(* IEC 61131-3 sources: std_i2980_v2.06_cp053/Source/IMM/ieccontrol/MoldHeightAdjust1 (part 3) *)

(* ---- ABAdjustPositionChange.pu ---- *)
(*
@h    ! WARNING !
@h    The Kemro K2 system (including software) only meets category B according to EN 954-1,
@h    thus it is not intended for usage in safety-relevant control applications in the field
@h    of personal safety (e.g. emergency stop).
@h    To implement potentially necessary safety-relevant control tasks, always use additional
@h    external safety devices that are intended for the particular purpose, and meet the necessary
@h    functional safety.
@h    For further information see EN 954-1 (EN ISO 13849-1) and/or the K2-x00 user manual, chapter
@h    "CE conformity, directives and standards".

This algo sends the mold height to a specified position by controlling the
Mold Height Movements.
*)

IMPORT_OVER_LISTFILE
 SET_ALARM
, cMoveFwd
, cMoveMoldHeight
, cMoveBwd
, tsMoldHeightPositions
, tsEndpointMonitor
, tevStartRequest
, tsDeviceId
, tevStartRequestData
, FBStop
, FBCheckReady
, tnMovementDirection

END_IMPORT

ALGORITHM_BLOCK ABAdjustPositionChange #DUMMY_EDIT_BLOCK

SYSTEM_VAR
 sv_MoldHeightPositions : tsMoldHeightPositions;
 sv_MoldHeightEndpoints : tsEndpointMonitor;
 sv_rActMoldHeightPosition : REAL;
 sv_iThisStepsSetImpulses : UDINT;
 sv_rDistancePerImpulse : REAL;
END_VAR

SYSTEM_OBJECT
 evStartRequest : tevStartRequest;
 erMoldHeightAdjustAborted : ALARM;
 erMoldHeightAdjustFinished : ALARM;
END_OBJECT

(*
This algo controls the mold height automatic position change:
- A desired position is set on the hmi. By starting the automatic mold height adjustment this algo is called.
- The desired position is translated into a number of increments and direction to move to.
- The movement is started until the position reached flags are set by the movements of MoldHeight1.
- The ready flag is set and the algo won't be called any more.
*)

ALGORITHM aRun

VAR_INPUT
 bStop : BOOL;
END_VAR

VAR_OUTPUT
 bReady : BOOL;
END_VAR

VAR_INPUT
 DeviceIdMoldHeight : tsDeviceId;
END_VAR

VAR
 iTempImpulses : INT;
 evStartRequestData : tevStartRequestData;
 fbStop : FBStop;
 fbCheckReady : FBCheckReady;
 MovementDirection : tnMovementDirection;
END_VAR

(* IecGraph-Code *)

(* init step *)
INITIAL_STEP START:
END_STEP

(* steps *)
STEP PREPARE_MOVEMENT:
aPrepareMovement (P);
END_STEP

STEP MOVE:
AReset (P);
END_STEP

ACTION AReset: #BEGIN_EDIT_BLOCK
sv_MoldHeightEndpoints.bPositionForStepReached := FALSE;

;#END_EDIT_BLOCK END_ACTION (*AReset*)
STEP MOVE_FWD_TO_POS:
aMoveFwdToPos (P);
aCheckFwdReady (N);
END_STEP

STEP MOVE_BWD_TO_POS:
aMoveBwdToPos (P);
aCheckBwdReady (N);
END_STEP

STEP READY:
ResetMovementFlags (P);
END_STEP

ACTION ResetMovementFlags: #BEGIN_EDIT_BLOCK
IF bStop THEN
    //stop active device
    fbStop(DeviceId := DeviceIdMoldHeight);
END_IF;

IF sv_MoldHeightEndpoints.bPositionForStepReached THEN
    SET_ALARM(erMoldHeightAdjustFinished);
ELSE
    SET_ALARM(erMoldHeightAdjustAborted);
END_IF;

bReady := TRUE;

;#END_EDIT_BLOCK END_ACTION (*ResetMovementFlags*)

(* transitions *)
GO_ON_TRANSITION StartTrans FROM START TO PREPARE_MOVEMENT :=  #BEGIN_EDIT_BLOCK
TRUE
;#END_EDIT_BLOCK
END_TRANSITION

GO_ON_TRANSITION TAdjust FROM PREPARE_MOVEMENT TO MOVE :=  #BEGIN_EDIT_BLOCK
iTempImpulses <> 0
;#END_EDIT_BLOCK
END_TRANSITION

GO_ON_TRANSITION TNoAdjustNeeded FROM PREPARE_MOVEMENT TO READY :=  #BEGIN_EDIT_BLOCK
iTempImpulses = 0
;#END_EDIT_BLOCK
END_TRANSITION

GO_ON_TRANSITION CheckMovementDirection1 FROM MOVE TO MOVE_FWD_TO_POS :=  #BEGIN_EDIT_BLOCK
MovementDirection = nForward
;#END_EDIT_BLOCK
END_TRANSITION

TRANSITION CheckMovementFinished1 FROM MOVE_FWD_TO_POS TO READY :=  #BEGIN_EDIT_BLOCK
fbCheckReady.bReady OR bStop
;#END_EDIT_BLOCK
END_TRANSITION

GO_ON_TRANSITION CheckMovementDirection2 FROM MOVE TO MOVE_BWD_TO_POS :=  #BEGIN_EDIT_BLOCK
MovementDirection = nBackward
;#END_EDIT_BLOCK
END_TRANSITION

TRANSITION CheckMovementFinished2 FROM MOVE_BWD_TO_POS TO READY :=  #BEGIN_EDIT_BLOCK
fbCheckReady.bReady OR bStop
;#END_EDIT_BLOCK
END_TRANSITION

TRANSITION TLoopBack FROM READY TO START :=  #BEGIN_EDIT_BLOCK
TRUE
;#END_EDIT_BLOCK
END_TRANSITION

(* end IecGraph-Code *)
(* sfc-code *)

(* stand alone actions *)
ACTION aMoveFwdToPos: #BEGIN_EDIT_BLOCK
(*@ MoldHeightAdjustN.ABAdjustPositionChange.aMoveFwdToPos.Start the mold height forward movement.*)
evStartRequestData.DeviceId := DeviceIdMoldHeight;
evStartRequestData.MoveDir := cMoveFwd;
evStartRequestData.MoveId := cMoveFwd;
SET_EVENT(evStartRequest, evStartRequestData);

;#END_EDIT_BLOCK END_ACTION (*aMoveFwdToPos*)
ACTION aMoveBwdToPos: #BEGIN_EDIT_BLOCK
(*@ MoldHeightAdjustN.ABAdjustPositionChange.aMoveBwdToPos.Start the mold height backwar movement.*)
evStartRequestData.DeviceId := DeviceIdMoldHeight;
evStartRequestData.MoveDir := cMoveBwd;
evStartRequestData.MoveId := cMoveBwd;
SET_EVENT(evStartRequest, evStartRequestData);

;#END_EDIT_BLOCK END_ACTION (*aMoveBwdToPos*)
ACTION aPrepareMovement: #BEGIN_EDIT_BLOCK

(*@ MoldHeightAdjustN.ABAdjustPositionChange.aPrepareMovement.Reset the CalcFinished and AutoAdjustFinished flag
                                                for normal operation.*)
bReady := FALSE;

(*@ MoldHeightAdjustN.ABAdjustPositionChange.aPrepareMovement.Calculate the number of Impulses the mold height
                                                should move like this:
                                                Distance = Actual Position - MoveTo Position;
                                                Impulses To Move = Distance / Distance per Impulse*)
IF sv_rDistancePerImpulse > 0.0 THEN
   //avoid division by zero
   iTempImpulses := REAL_TO_INT((sv_rActMoldHeightPosition - sv_MoldHeightPositions.rMoveToMoldHeightPosition)/sv_rDistancePerImpulse);
ELSE
   iTempImpulses := 0;
END_IF;

(*@ MoldHeightAdjustN.ABAdjustPositionChange.aPrepareMovement.Check if the position as the same as the actual
                                                position and stop the movement if it so.
                                                Else check/set the direction. Negative number of Impulses to Move
                                                means Move Backward (If so, remove the negative sign of Impulses
                                                to Move.*)
IF iTempImpulses = 0 THEN
    bReady := TRUE;
ELSIF iTempImpulses < 0 THEN
    MovementDirection := nBackward;
    iTempImpulses := ABS(iTempImpulses);
ELSIF iTempImpulses > 0 THEN
    MovementDirection := nForward;
END_IF;

(*@ MoldHeightAdjustN.ABAdjustPositionChange.aPrepareMovement.Set the system variable for impulses to move*)
sv_iThisStepsSetImpulses := INT_TO_UDINT(iTempImpulses);

;#END_EDIT_BLOCK END_ACTION (*aPrepareMovement*)
ACTION aCheckFwdReady: #BEGIN_EDIT_BLOCK
(**************************************** WARNING ********************************************
 *** The KEBA Kemro K2 System including software is not intended for safety control tasks! ***
 ***                       For further information see Comment tab!                        ***
 *********************************************************************************************)

fbCheckReady(DeviceId := DeviceIdMoldHeight);

;#END_EDIT_BLOCK END_ACTION (*aCheckFwdReady*)
ACTION aCheckBwdReady: #BEGIN_EDIT_BLOCK
(**************************************** WARNING ********************************************
 *** The KEBA Kemro K2 System including software is not intended for safety control tasks! ***
 ***                       For further information see Comment tab!                        ***
 *********************************************************************************************)

fbCheckReady(DeviceId := DeviceIdMoldHeight);

;#END_EDIT_BLOCK END_ACTION (*aCheckBwdReady*)
(* end sfc-code *)

END_ALGORITHM

END_ALGORITHM_BLOCK

#END_OF_IEC_PART

@Puma @IecEditor 6 68 @Pou 25
@@@BEG_Comment@@@
@h    ! WARNING !
@h    The Kemro K2 system (including software) only meets category B according to EN 954-1,
@h    thus it is not intended for usage in safety-relevant control applications in the field
@h    of personal safety (e.g. emergency stop).
@h    To implement potentially necessary safety-relevant control tasks, always use additional
@h    external safety devices that are intended for the particular purpose, and meet the necessary
@h    functional safety.
@h    For further information see EN 954-1 (EN ISO 13849-1) and/or the K2-x00 user manual, chapter
@h    "CE conformity, directives and standards".

This algo sends the mold height to a specified position by controlling the
Mold Height Movements.
@@@END_Comment@@@

@BEG_Contents

@BEG_Func
@RT(17)FuncTreeContainer
1
@Var @RT(9)SET_ALARM @RT(0) @T @T @DERIVED 0 @F @RT(23)KEBA_STANDARD_PROCEDURE @F
@T
@BEG_Attrib
0 @RT(0) @RT(0)
@END_Attrib
1 1 @F @F @F @F

@END_Func

@BEG_Const
@RT(18)ConstTreeContainer
3
@Var @RT(8)cMoveFwd @RT(0) @T @F @DT @RT(4)DINT @RT(0) @T @T @BASIC 0 @F
@F @F
@T
@BEG_Attrib
0 @RT(2)12 @RT(16)movement forward
@END_Attrib
1 1 @F @F @F @F

@Var @RT(15)cMoveMoldHeight @RT(0) @T @F @DT @RT(4)DINT @RT(0) @T @T @BASIC 0 @F
@F @F
@T
@BEG_Attrib
0 @RT(2)29 @RT(23)movement of mold height
@END_Attrib
1 1 @F @F @F @F

@Var @RT(8)cMoveBwd @RT(0) @T @F @DT @RT(4)DINT @RT(0) @T @T @BASIC 0 @F
@F @F
@T
@BEG_Attrib
0 @RT(2)11 @RT(17)movement backward
@END_Attrib
1 1 @F @F @F @F

@END_Const

@BEG_Export

@BEG_Kind
@ALGORITHM_BLOCK @RT(22)ABAdjustPositionChange @STRUCTURED_TEXT
@RT(0) @RT(0) @RT(0)
@END_Kind

@BEG_Dcl
@RT(16)DclTreeContainer
8
@Var @RT(22)sv_MoldHeightPositions @RT(0) @T @T @DERIVED 0 @T @T @DT @RT(21)tsMoldHeightPositions @RT(0) @T @T @UNKNOWN 0 @F
@F @F
@T
@BEG_Attrib
3 @RT(0) @RT(0) @RT(0)
@END_Attrib
1 8 @F @F @F @F

@Var @RT(22)sv_MoldHeightEndpoints @RT(0) @T @T @DERIVED 0 @T @T @DT @RT(17)tsEndpointMonitor @RT(0) @T @T @UNKNOWN 0 @F
@F @F
@T
@BEG_Attrib
3 @RT(0) @RT(0) @RT(0)
@END_Attrib
1 8 @F @F @F @F

@Var @RT(25)sv_rActMoldHeightPosition @RT(0) @T @F @DT @RT(4)REAL @RT(0) @T @T @BASIC 0 @F
@F @F
@T
@BEG_Attrib
3 @RT(0) @RT(0) @RT(0)
@END_Attrib
1 8 @F @F @F @F

@Var @RT(24)sv_iThisStepsSetImpulses @RT(0) @T @F @DT @RT(5)UDINT @RT(0) @T @T @BASIC 0 @F
@F @F
@T
@BEG_Attrib
3 @RT(0) @RT(0) @RT(0)
@END_Attrib
1 8 @F @F @F @F

@Var @RT(22)sv_rDistancePerImpulse @RT(0) @T @F @DT @RT(4)REAL @RT(0) @T @T @BASIC 0 @F
@F @F
@T
@BEG_Attrib
3 @RT(0) @RT(0) @RT(0)
@END_Attrib
1 8 @F @F @F @F

@Var @RT(14)evStartRequest @RT(0) @T @T @DERIVED 0 @T @T @DT @RT(15)tevStartRequest @RT(0) @T @T @UNKNOWN 0 @F
@F @F
@T
@BEG_Attrib
3 @RT(0) @RT(0) @RT(0)
@END_Attrib
1 7 @F @F @F @F

@Var @RT(25)erMoldHeightAdjustAborted @RT(0) @T @F @DT @RT(5)ALARM @RT(0) @T @T @BASIC 0 @F
@F @F
@T
@BEG_Attrib
3 @RT(0) @RT(0) @RT(0)
@END_Attrib
1 7 @F @F @F @F

@Var @RT(26)erMoldHeightAdjustFinished @RT(0) @T @F @DT @RT(5)ALARM @RT(0) @T @T @BASIC 0 @F
@F @F
@T
@BEG_Attrib
3 @RT(0) @RT(0) @RT(0)
@END_Attrib
1 7 @F @F @F @F

@END_Dcl

@END_Export

@BEG_Body

1

@BEG_Export

@BEG_Algo
@ALGORITHM @RT(4)aRun @SEQUENTIAL_FLOW_CHART
@RT(0) @RT(0) @RT(0) @F @F
@END_Algo

@BEG_Dcl
@RT(16)DclTreeContainer
8
@Var @RT(5)bStop @RT(0) @T @F @DT @RT(4)BOOL @RT(0) @T @T @BASIC 0 @F
@F @F
@T
@BEG_Attrib
3 @RT(0) @RT(0) @RT(0)
@END_Attrib
1 1 @F @F @F @F

@Var @RT(6)bReady @RT(0) @T @F @DT @RT(4)BOOL @RT(0) @T @T @BASIC 0 @F
@F @F
@T
@BEG_Attrib
3 @RT(0) @RT(0) @RT(0)
@END_Attrib
1 3 @F @F @F @F

@Var @RT(18)DeviceIdMoldHeight @RT(0) @T @T @DERIVED 0 @T @T @DT @RT(10)tsDeviceId @RT(0) @T @T @UNKNOWN 0 @F
@F @F
@T
@BEG_Attrib
3 @RT(0) @RT(0) @RT(0)
@END_Attrib
1 1 @F @F @F @F

@Var @RT(13)iTempImpulses @RT(0) @T @F @DT @RT(3)INT @RT(0) @T @T @BASIC 0 @F
@F @F
@T
@BEG_Attrib
3 @RT(0) @RT(0) @RT(0)
@END_Attrib
1 0 @F @F @F @F

@Var @RT(18)evStartRequestData @RT(0) @T @T @DERIVED 0 @T @T @DT @RT(19)tevStartRequestData @RT(0) @T @T @UNKNOWN 0 @F
@F @F
@T
@BEG_Attrib
3 @RT(0) @RT(0) @RT(0)
@END_Attrib
1 0 @F @F @F @F

@Var @RT(6)fbStop @RT(0) @T @T @DERIVED 0 @T @T @DT @RT(6)FBStop @RT(0) @T @T @UNKNOWN 0 @F
@F @F
@T
@BEG_Attrib
3 @RT(0) @RT(0) @RT(0)
@END_Attrib
1 0 @F @F @F @F

@Var @RT(12)fbCheckReady @RT(0) @T @T @DERIVED 0 @T @T @DT @RT(12)FBCheckReady @RT(0) @T @T @UNKNOWN 0 @F
@F @F
@T
@BEG_Attrib
3 @RT(0) @RT(0) @RT(0)
@END_Attrib
1 0 @F @F @F @F

@Var @RT(17)MovementDirection @RT(0) @T @T @DERIVED 0 @T @T @DT @RT(19)tnMovementDirection @RT(0) @T @T @UNKNOWN 0 @F
@F @F
@T
@BEG_Attrib
3 @RT(0) @RT(0) @RT(0)
@END_Attrib
1 0 @F @F @F @F

@END_Dcl

@END_Export

@BEG_SfcBody
17 12 14

@BEG_SfcData 2
@StepSeq @RT(4)sseq @F 1
@Loop @RT(4)loop @F 2
@StepSeq @RT(3)seq @F 7
@Step @RT(5)START @F @T @F @F @RT(0) @F
@AcbCont @RT(7)unnamed @F 0

@Trans @RT(10)StartTrans @F @T @F @F @T @F @TL(2)
TRUE

@RT(6)Trans1 @F
@Step @RT(16)PREPARE_MOVEMENT @F @F @F @F @RT(0) @F
@AcbCont @RT(7)unnamed @F 1
@Acb @RT(16)aPrepareMovement @F @F @RT(1)P @RT(0) @F @F @T @F

@AltBranch @RT(3)alt @F 2
@TransSeq @RT(4)tseq @F 1
@Trans @RT(7)TAdjust @F @T @F @F @T @F @TL(2)
iTempImpulses <> 0

@RT(6)Trans2 @F

@TransSeq @RT(4)tseq @F 2
@Trans @RT(15)TNoAdjustNeeded @F @T @F @F @T @F @TL(2)
iTempImpulses = 0

@RT(7)Trans13 @F
@Goto @RT(5)READY @F @F

@Step @RT(4)MOVE @F @F @F @F @RT(0) @F
@AcbCont @RT(7)unnamed @F 1
@Acb @RT(6)AReset @F @T @RT(1)P @RT(0) @F @F @T @TL(2)
sv_MoldHeightEndpoints.bPositionForStepReached := FALSE;

@F

@AltBranch @RT(3)alt @F 2
@TransSeq @RT(4)tseq @F 3
@Trans @RT(23)CheckMovementDirection1 @F @T @F @F @T @F @TL(2)
MovementDirection = nForward

@RT(6)Trans3 @F
@Step @RT(15)MOVE_FWD_TO_POS @F @F @F @F @RT(0) @F
@AcbCont @RT(7)unnamed @F 2
@Acb @RT(13)aMoveFwdToPos @F @F @RT(1)P @RT(0) @F @F @T @F
@Acb @RT(14)aCheckFwdReady @F @F @RT(1)N @RT(0) @F @F @F @F

@Trans @RT(22)CheckMovementFinished1 @F @T @F @F @T @T @TL(2)
fbCheckReady.bReady OR bStop

@RT(6)Trans5 @F

@TransSeq @RT(4)tseq @F 3
@Trans @RT(23)CheckMovementDirection2 @F @T @F @F @T @F @TL(2)
MovementDirection = nBackward

@RT(6)Trans4 @F
@Step @RT(15)MOVE_BWD_TO_POS @F @F @F @F @RT(0) @F
@AcbCont @RT(7)unnamed @F 2
@Acb @RT(13)aMoveBwdToPos @F @F @RT(1)P @RT(0) @F @F @F @F
@Acb @RT(14)aCheckBwdReady @F @F @RT(1)N @RT(0) @F @F @F @F

@Trans @RT(22)CheckMovementFinished2 @F @T @F @F @T @T @TL(2)
fbCheckReady.bReady OR bStop

@RT(6)Trans5 @F

@Step @RT(5)READY @F @F @T @F @RT(0) @F
@AcbCont @RT(7)unnamed @F 1
@Acb @RT(18)ResetMovementFlags @F @T @RT(1)P @RT(0) @F @F @T @TL(13)
IF bStop THEN
    //stop active device
    fbStop(DeviceId := DeviceIdMoldHeight);
END_IF;

IF sv_MoldHeightEndpoints.bPositionForStepReached THEN
    SET_ALARM(erMoldHeightAdjustFinished);
ELSE
    SET_ALARM(erMoldHeightAdjustAborted);
END_IF;

bReady := TRUE;

@F

@Trans @RT(9)TLoopBack @F @T @T @T @T @T @TL(2)
TRUE

@RT(6)Trans7 @F

@END_SfcData
@SaActions 5
@SaText @RT(13)aMoveFwdToPos 1 @TL(6)
(*@ MoldHeightAdjustN.ABAdjustPositionChange.aMoveFwdToPos.Start the mold height forward movement.*)
evStartRequestData.DeviceId := DeviceIdMoldHeight;
evStartRequestData.MoveDir := cMoveFwd;
evStartRequestData.MoveId := cMoveFwd;
SET_EVENT(evStartRequest, evStartRequestData);

@SaText @RT(13)aMoveBwdToPos 1 @TL(6)
(*@ MoldHeightAdjustN.ABAdjustPositionChange.aMoveBwdToPos.Start the mold height backwar movement.*)
evStartRequestData.DeviceId := DeviceIdMoldHeight;
evStartRequestData.MoveDir := cMoveBwd;
evStartRequestData.MoveId := cMoveBwd;
SET_EVENT(evStartRequest, evStartRequestData);

@SaText @RT(16)aPrepareMovement 1 @TL(33)

(*@ MoldHeightAdjustN.ABAdjustPositionChange.aPrepareMovement.Reset the CalcFinished and AutoAdjustFinished flag
                                                for normal operation.*)
bReady := FALSE;

(*@ MoldHeightAdjustN.ABAdjustPositionChange.aPrepareMovement.Calculate the number of Impulses the mold height
                                                should move like this:
                                                Distance = Actual Position - MoveTo Position;
                                                Impulses To Move = Distance / Distance per Impulse*)
IF sv_rDistancePerImpulse > 0.0 THEN
   //avoid division by zero
   iTempImpulses := REAL_TO_INT((sv_rActMoldHeightPosition - sv_MoldHeightPositions.rMoveToMoldHeightPosition)/sv_rDistancePerImpulse);
ELSE
   iTempImpulses := 0;
END_IF;

(*@ MoldHeightAdjustN.ABAdjustPositionChange.aPrepareMovement.Check if the position as the same as the actual
                                                position and stop the movement if it so.
                                                Else check/set the direction. Negative number of Impulses to Move
                                                means Move Backward (If so, remove the negative sign of Impulses
                                                to Move.*)
IF iTempImpulses = 0 THEN
    bReady := TRUE;
ELSIF iTempImpulses < 0 THEN
    MovementDirection := nBackward;
    iTempImpulses := ABS(iTempImpulses);
ELSIF iTempImpulses > 0 THEN
    MovementDirection := nForward;
END_IF;

(*@ MoldHeightAdjustN.ABAdjustPositionChange.aPrepareMovement.Set the system variable for impulses to move*)
sv_iThisStepsSetImpulses := INT_TO_UDINT(iTempImpulses);

@SaText @RT(14)aCheckFwdReady 1 @TL(7)
(**************************************** WARNING ********************************************
 *** The KEBA Kemro K2 System including software is not intended for safety control tasks! ***
 ***                       For further information see Comment tab!                        ***
 *********************************************************************************************)

fbCheckReady(DeviceId := DeviceIdMoldHeight);

@SaText @RT(14)aCheckBwdReady 1 @TL(7)
(**************************************** WARNING ********************************************
 *** The KEBA Kemro K2 System including software is not intended for safety control tasks! ***
 ***                       For further information see Comment tab!                        ***
 *********************************************************************************************)

fbCheckReady(DeviceId := DeviceIdMoldHeight);

@SaTrans 0
@SaExits 0
@END_SfcBody

@@@BEG_Comment@@@
@TL(5)
This algo controls the mold height automatic position change:
- A desired position is set on the hmi. By starting the automatic mold height adjustment this algo is called.
- The desired position is translated into a number of increments and direction to move to.
- The movement is started until the position reached flags are set by the movements of MoldHeight1.
- The ready flag is set and the algo won't be called any more.
@@@END_Comment@@@
@END_Body

@END_Contents

(* ---- ABAdjustPosSetTonnage.pu ---- *)
(*
@h    ! WARNING !
@h    The Kemro K2 system (including software) only meets category B according to EN 954-1,
@h    thus it is not intended for usage in safety-relevant control applications in the field
@h    of personal safety (e.g. emergency stop).
@h    To implement potentially necessary safety-relevant control tasks, always use additional
@h    external safety devices that are intended for the particular purpose, and meet the necessary
@h    functional safety.
@h    For further information see EN 954-1 (EN ISO 13849-1) and/or the K2-x00 user manual, chapter
@h    "CE conformity, directives and standards".

This algo sends the mold height to a specified position by controlling the
Mold Height Movements.
*)

IMPORT_OVER_LISTFILE
 SET_ALARM
, cMoveFwd
, cMoveMoldHeight
, cMoveBwd
, tsEndpointMonitor
, tevStartRequest
, KAPPL_LintabData
, tsClampForces
, ABCalculateMoldHeightImpulses
, tsDeviceId
, tevStartRequestData
, FBStop
, FBCheckReady
, FBCheckPosReached
, tnMovementDirection

END_IMPORT

ALGORITHM_BLOCK ABAdjustPosSetTonnage #DUMMY_EDIT_BLOCK

SYSTEM_VAR
 sv_MoldHeightEndpoints : tsEndpointMonitor;
 sv_iThisStepsSetImpulses : UDINT;
 sv_ClampForceLintabImpulses : KAPPL_LintabData;
 sv_iThisStepsActImpulses : UDINT;
 sv_ClampForce : tsClampForces;
END_VAR

SYSTEM_OBJECT
 evStartRequest : tevStartRequest;
 erMoldHeightAdjustAborted : ALARM;
 erMoldHeightAdjustFinished : ALARM;
 erMoldHeightAdjustMoldNotOpen : ALARM;
END_OBJECT

VAR
 abCalculateMoldHeightImpulses : ABCalculateMoldHeightImpulses;
END_VAR

(*
This algo controls the mold height automatic position change:
- A desired position is set on the hmi. By starting the automatic mold height adjustment this algo is called.
- The desired position is translated into a number of increments and direction to move to.
- The movement is started until the position reached flags are set by the movements of MoldHeight1.
- The ready flag is set and the algo won't be called any more.
*)

ALGORITHM aRun

VAR_INPUT
 bStop : BOOL;
END_VAR

VAR_OUTPUT
 bReady : BOOL;
END_VAR

VAR_INPUT
 DeviceIdMoldHeight : tsDeviceId;
 DeviceIdMold : tsDeviceId;
END_VAR

VAR
 iTempImpulses : DINT;
 evStartRequestData : tevStartRequestData;
 fbStop : FBStop;
 fbCheckReady : FBCheckReady;
 fbCheckPosReached : FBCheckPosReached;
 bMoldOpen : BOOL;
 iImpulseActPos : DINT (* Actual Impulse position calculated from clamping force *);
 MovementDirection : tnMovementDirection;
END_VAR

(* IecGraph-Code *)

(* init step *)
INITIAL_STEP START:
END_STEP

(* steps *)
STEP PREPARE_MOVEMENT:
ACheckMoldBackward (P);
aPrepareMovement (P);
END_STEP

STEP MOVE:
AReset (P);
END_STEP

ACTION AReset: #BEGIN_EDIT_BLOCK
sv_MoldHeightEndpoints.bPositionForStepReached := FALSE;

;#END_EDIT_BLOCK END_ACTION (*AReset*)
STEP MOVE_FWD_TO_POS:
aMoveFwdToPos (P);
aCheckFwdReady (N);
END_STEP

STEP MOVE_BWD_TO_POS:
aMoveBwdToPos (P);
aCheckBwdReady (N);
END_STEP

STEP READY:
AUpdateClampForce (P);
ResetMovementFlags (P);
END_STEP

ACTION ResetMovementFlags: #BEGIN_EDIT_BLOCK
IF bStop THEN
    //stop active device
    fbStop(DeviceId := DeviceIdMoldHeight);
END_IF;

IF NOT bMoldOpen THEN
    SET_ALARM(erMoldHeightAdjustMoldNotOpen);
END_IF;

IF sv_MoldHeightEndpoints.bPositionForStepReached THEN
    SET_ALARM(erMoldHeightAdjustFinished);
ELSE
    SET_ALARM(erMoldHeightAdjustAborted);
END_IF;

bReady := TRUE;

;#END_EDIT_BLOCK END_ACTION (*ResetMovementFlags*)

(* transitions *)
GO_ON_TRANSITION StartTrans FROM START TO PREPARE_MOVEMENT :=  #BEGIN_EDIT_BLOCK
TRUE
;#END_EDIT_BLOCK
END_TRANSITION

GO_ON_TRANSITION TAdjust FROM PREPARE_MOVEMENT TO MOVE :=  #BEGIN_EDIT_BLOCK
bMoldOpen AND iTempImpulses <> 0
;#END_EDIT_BLOCK
END_TRANSITION

GO_ON_TRANSITION TNoAdjustNeeded FROM PREPARE_MOVEMENT TO READY :=  #BEGIN_EDIT_BLOCK
bMoldOpen AND iTempImpulses = 0
;#END_EDIT_BLOCK
END_TRANSITION

GO_ON_TRANSITION TMoldNotOpen FROM PREPARE_MOVEMENT TO READY :=  #BEGIN_EDIT_BLOCK
NOT bMoldOpen
;#END_EDIT_BLOCK
END_TRANSITION

GO_ON_TRANSITION CheckMovementDirection1 FROM MOVE TO MOVE_FWD_TO_POS :=  #BEGIN_EDIT_BLOCK
MovementDirection = nForward
;#END_EDIT_BLOCK
END_TRANSITION

TRANSITION CheckMovementFinished1 FROM MOVE_FWD_TO_POS TO READY :=  #BEGIN_EDIT_BLOCK
fbCheckReady.bReady OR bStop
;#END_EDIT_BLOCK
END_TRANSITION

GO_ON_TRANSITION CheckMovementDirection2 FROM MOVE TO MOVE_BWD_TO_POS :=  #BEGIN_EDIT_BLOCK
MovementDirection = nBackward
;#END_EDIT_BLOCK
END_TRANSITION

TRANSITION CheckMovementFinished2 FROM MOVE_BWD_TO_POS TO READY :=  #BEGIN_EDIT_BLOCK
fbCheckReady.bReady OR bStop
;#END_EDIT_BLOCK
END_TRANSITION

TRANSITION TLoopBack FROM READY TO START :=  #BEGIN_EDIT_BLOCK
TRUE
;#END_EDIT_BLOCK
END_TRANSITION

(* end IecGraph-Code *)
(* sfc-code *)

(* stand alone actions *)
ACTION aMoveFwdToPos: #BEGIN_EDIT_BLOCK
(*@ MoldHeightAdjustN.ABAdjustPositionChange.aMoveFwdToPos.Start the mold height forward movement.*)
evStartRequestData.DeviceId := DeviceIdMoldHeight;
evStartRequestData.MoveDir := cMoveFwd;
evStartRequestData.MoveId := cMoveFwd;
SET_EVENT(evStartRequest, evStartRequestData);

;#END_EDIT_BLOCK END_ACTION (*aMoveFwdToPos*)
ACTION aMoveBwdToPos: #BEGIN_EDIT_BLOCK
(*@ MoldHeightAdjustN.ABAdjustPositionChange.aMoveBwdToPos.Start the mold height backwar movement.*)
evStartRequestData.DeviceId := DeviceIdMoldHeight;
evStartRequestData.MoveDir := cMoveBwd;
evStartRequestData.MoveId := cMoveBwd;
SET_EVENT(evStartRequest, evStartRequestData);

;#END_EDIT_BLOCK END_ACTION (*aMoveBwdToPos*)
ACTION aPrepareMovement: #BEGIN_EDIT_BLOCK
(**************************************** WARNING ********************************************
 *** The KEBA Kemro K2 System including software is not intended for safety control tasks! ***
 ***                       For further information see Comment tab!                        ***
 *********************************************************************************************)

// Reset the CalcFinished and AutoAdjustFinished flag
// for normal operation.
bReady := FALSE;
iTempImpulses := 0;

abCalculateMoldHeightImpulses.aInit(Lintab := sv_ClampForceLintabImpulses);
abCalculateMoldHeightImpulses.aCalc(rForce := sv_ClampForce.rActualClampForce);
iImpulseActPos := abCalculateMoldHeightImpulses.aCalc.iImpulses;

abCalculateMoldHeightImpulses.aCalc(rForce := sv_ClampForce.rSetClampForce);
iTempImpulses := abCalculateMoldHeightImpulses.aCalc.iImpulses - iImpulseActPos;
//abCalculateMoldHeightImpulses.aCalc( rActualForce:= sv_ClampForce.rActualClampForce, rSetForce:= sv_ClampForce.rSetClampForce);
//iTempImpulses := abCalculateMoldHeightImpulses.aCalc.iImpulses;

IF iTempImpulses = 0 THEN
    bReady := TRUE;
ELSIF iTempImpulses < 0 THEN
    MovementDirection := nBackward;
    iTempImpulses := ABS(iTempImpulses);
ELSIF iTempImpulses > 0 THEN
    MovementDirection := nForward;
END_IF;

// Set the system variable for impulses to move
sv_iThisStepsSetImpulses := DINT_TO_UDINT(iTempImpulses);
sv_iThisStepsActImpulses := 0;

;#END_EDIT_BLOCK END_ACTION (*aPrepareMovement*)
ACTION aCheckFwdReady: #BEGIN_EDIT_BLOCK
(**************************************** WARNING ********************************************
 *** The KEBA Kemro K2 System including software is not intended for safety control tasks! ***
 ***                       For further information see Comment tab!                        ***
 *********************************************************************************************)

fbCheckReady(DeviceId := DeviceIdMoldHeight);

;#END_EDIT_BLOCK END_ACTION (*aCheckFwdReady*)
ACTION aCheckBwdReady: #BEGIN_EDIT_BLOCK
(**************************************** WARNING ********************************************
 *** The KEBA Kemro K2 System including software is not intended for safety control tasks! ***
 ***                       For further information see Comment tab!                        ***
 *********************************************************************************************)

fbCheckReady(DeviceId := DeviceIdMoldHeight);

;#END_EDIT_BLOCK END_ACTION (*aCheckBwdReady*)
ACTION ACheckMoldBackward: #BEGIN_EDIT_BLOCK

fbCheckPosReached(DeviceId := DeviceIdMold,
                  MoveDir := cMoveBwd,
                  MoveId := cMoveBwdForMHAdjust,
                  bPosReached => bMoldOpen);

;#END_EDIT_BLOCK END_ACTION (*ACheckMoldBackward*)
ACTION AUpdateClampForce: #BEGIN_EDIT_BLOCK
(**************************************** WARNING ********************************************
 *** The KEBA Kemro K2 System including software is not intended for safety control tasks! ***
 ***                       For further information see Comment tab!                        ***
 *********************************************************************************************)

// calculate actual new clamping foce at end of movement
abCalculateMoldHeightImpulses.aInit(Lintab := sv_ClampForceLintabImpulses);
IF MovementDirection = nForward THEN
    abCalculateMoldHeightImpulses.aCalcInv(iImpulses := iImpulseActPos + UDINT_TO_DINT(sv_iThisStepsActImpulses));
ELSE
    abCalculateMoldHeightImpulses.aCalcInv(iImpulses := iImpulseActPos - UDINT_TO_DINT(sv_iThisStepsActImpulses));
END_IF;

sv_ClampForce.rActualClampForce := abCalculateMoldHeightImpulses.aCalcInv.rForce;

;#END_EDIT_BLOCK END_ACTION (*AUpdateClampForce*)
(* end sfc-code *)

END_ALGORITHM

END_ALGORITHM_BLOCK

#END_OF_IEC_PART

@Puma @IecEditor 6 30 @Pou 25
@@@BEG_Comment@@@
@h    ! WARNING !
@h    The Kemro K2 system (including software) only meets category B according to EN 954-1,
@h    thus it is not intended for usage in safety-relevant control applications in the field
@h    of personal safety (e.g. emergency stop).
@h    To implement potentially necessary safety-relevant control tasks, always use additional
@h    external safety devices that are intended for the particular purpose, and meet the necessary
@h    functional safety.
@h    For further information see EN 954-1 (EN ISO 13849-1) and/or the K2-x00 user manual, chapter
@h    "CE conformity, directives and standards".

This algo sends the mold height to a specified position by controlling the
Mold Height Movements.
@@@END_Comment@@@

@BEG_Contents

@BEG_Func
@RT(17)FuncTreeContainer
1
@Var @RT(9)SET_ALARM @RT(0) @T @T @DERIVED 0 @F @RT(23)KEBA_STANDARD_PROCEDURE @F
@T
@BEG_Attrib
0 @RT(0) @RT(0)
@END_Attrib
1 1 @F @F @F @F

@END_Func

@BEG_Const
@RT(18)ConstTreeContainer
3
@Var @RT(8)cMoveFwd @RT(0) @T @F @DT @RT(4)DINT @RT(0) @T @T @BASIC 0 @F
@F @F
@T
@BEG_Attrib
0 @RT(2)12 @RT(16)movement forward
@END_Attrib
1 1 @F @F @F @F

@Var @RT(15)cMoveMoldHeight @RT(0) @T @F @DT @RT(4)DINT @RT(0) @T @T @BASIC 0 @F
@F @F
@T
@BEG_Attrib
0 @RT(2)29 @RT(23)movement of mold height
@END_Attrib
1 1 @F @F @F @F

@Var @RT(8)cMoveBwd @RT(0) @T @F @DT @RT(4)DINT @RT(0) @T @T @BASIC 0 @F
@F @F
@T
@BEG_Attrib
0 @RT(2)11 @RT(17)movement backward
@END_Attrib
1 1 @F @F @F @F

@END_Const

@BEG_Export

@BEG_Kind
@ALGORITHM_BLOCK @RT(21)ABAdjustPosSetTonnage @STRUCTURED_TEXT
@RT(0) @RT(0) @RT(0)
@END_Kind

@BEG_Dcl
@RT(16)DclTreeContainer
10
@Var @RT(22)sv_MoldHeightEndpoints @RT(0) @T @T @DERIVED 0 @T @T @DT @RT(17)tsEndpointMonitor @RT(0) @T @T @UNKNOWN 0 @F
@F @F
@T
@BEG_Attrib
3 @RT(0) @RT(0) @RT(0)
@END_Attrib
1 8 @F @F @F @F

@Var @RT(24)sv_iThisStepsSetImpulses @RT(0) @T @F @DT @RT(5)UDINT @RT(0) @T @T @BASIC 0 @F
@F @F
@T
@BEG_Attrib
3 @RT(0) @RT(0) @RT(0)
@END_Attrib
1 8 @F @F @F @F

@Var @RT(14)evStartRequest @RT(0) @T @T @DERIVED 0 @T @T @DT @RT(15)tevStartRequest @RT(0) @T @T @UNKNOWN 0 @F
@F @F
@T
@BEG_Attrib
3 @RT(0) @RT(0) @RT(0)
@END_Attrib
1 7 @F @F @F @F

@Var @RT(25)erMoldHeightAdjustAborted @RT(0) @T @F @DT @RT(5)ALARM @RT(0) @T @T @BASIC 0 @F
@F @F
@T
@BEG_Attrib
3 @RT(0) @RT(0) @RT(0)
@END_Attrib
1 7 @F @F @F @F

@Var @RT(26)erMoldHeightAdjustFinished @RT(0) @T @F @DT @RT(5)ALARM @RT(0) @T @T @BASIC 0 @F
@F @F
@T
@BEG_Attrib
3 @RT(0) @RT(0) @RT(0)
@END_Attrib
1 7 @F @F @F @F

@Var @RT(27)sv_ClampForceLintabImpulses @RT(0) @T @T @RENAMED 0 @T @T @DT @RT(16)KAPPL_LintabData @RT(0) @T @T @UNKNOWN 0 @F
@F @F
@T
@BEG_Attrib
3 @RT(0) @RT(0) @RT(0)
@END_Attrib
1 8 @F @F @F @F

@Var @RT(29)erMoldHeightAdjustMoldNotOpen @RT(0) @T @T @RENAMED 0 @T @T @DT @RT(5)ALARM @RT(0) @T @T @BASIC 0 @F
@F @F
@T
@BEG_Attrib
3 @RT(0) @RT(0) @RT(0)
@END_Attrib
1 7 @F @F @F @F

@Var @RT(24)sv_iThisStepsActImpulses @RT(0) @T @T @RENAMED 0 @T @T @DT @RT(5)UDINT @RT(0) @T @T @BASIC 0 @F
@F @F
@T
@BEG_Attrib
3 @RT(0) @RT(0) @RT(0)
@END_Attrib
1 8 @F @F @F @F

@Var @RT(13)sv_ClampForce @RT(0) @T @T @DERIVED 0 @T @T @DT @RT(13)tsClampForces @RT(0) @T @T @UNKNOWN 0 @F
@F @F
@T
@BEG_Attrib
3 @RT(0) @RT(0) @RT(0)
@END_Attrib
1 8 @F @F @F @F

@Var @RT(29)abCalculateMoldHeightImpulses @RT(0) @T @T @DERIVED 0 @T @T @DT @RT(29)ABCalculateMoldHeightImpulses @RT(0) @T @T @UNKNOWN 0 @F
@F @F
@T
@BEG_Attrib
3 @RT(0) @RT(0) @RT(0)
@END_Attrib
1 0 @F @F @F @F

@END_Dcl

@END_Export

@BEG_Body

1

@BEG_Export

@BEG_Algo
@ALGORITHM @RT(4)aRun @SEQUENTIAL_FLOW_CHART
@RT(0) @RT(0) @RT(0) @F @F
@END_Algo

@BEG_Dcl
@RT(16)DclTreeContainer
12
@Var @RT(5)bStop @RT(0) @T @F @DT @RT(4)BOOL @RT(0) @T @T @BASIC 0 @F
@F @F
@T
@BEG_Attrib
3 @RT(0) @RT(0) @RT(0)
@END_Attrib
1 1 @F @F @F @F

@Var @RT(6)bReady @RT(0) @T @F @DT @RT(4)BOOL @RT(0) @T @T @BASIC 0 @F
@F @F
@T
@BEG_Attrib
3 @RT(0) @RT(0) @RT(0)
@END_Attrib
1 3 @F @F @F @F

@Var @RT(18)DeviceIdMoldHeight @RT(0) @T @T @DERIVED 0 @T @T @DT @RT(10)tsDeviceId @RT(0) @T @T @UNKNOWN 0 @F
@F @F
@T
@BEG_Attrib
3 @RT(0) @RT(0) @RT(0)
@END_Attrib
1 1 @F @F @F @F

@Var @RT(12)DeviceIdMold @RT(0) @T @T @DERIVED 0 @T @T @DT @RT(10)tsDeviceId @RT(0) @T @T @UNKNOWN 0 @F
@F @F
@T
@BEG_Attrib
3 @RT(0) @RT(0) @RT(0)
@END_Attrib
1 1 @F @F @F @F

@Var @RT(13)iTempImpulses @RT(0) @T @F @DT @RT(4)DINT @RT(0) @T @T @BASIC 0 @F
@F @F
@T
@BEG_Attrib
3 @RT(0) @RT(0) @RT(0)
@END_Attrib
1 0 @F @F @F @F

@Var @RT(18)evStartRequestData @RT(0) @T @T @DERIVED 0 @T @T @DT @RT(19)tevStartRequestData @RT(0) @T @T @UNKNOWN 0 @F
@F @F
@T
@BEG_Attrib
3 @RT(0) @RT(0) @RT(0)
@END_Attrib
1 0 @F @F @F @F

@Var @RT(6)fbStop @RT(0) @T @T @DERIVED 0 @T @T @DT @RT(6)FBStop @RT(0) @T @T @UNKNOWN 0 @F
@F @F
@T
@BEG_Attrib
3 @RT(0) @RT(0) @RT(0)
@END_Attrib
1 0 @F @F @F @F

@Var @RT(12)fbCheckReady @RT(0) @T @T @DERIVED 0 @T @T @DT @RT(12)FBCheckReady @RT(0) @T @T @UNKNOWN 0 @F
@F @F
@T
@BEG_Attrib
3 @RT(0) @RT(0) @RT(0)
@END_Attrib
1 0 @F @F @F @F

@Var @RT(17)fbCheckPosReached @RT(0) @T @T @DERIVED 0 @T @T @DT @RT(17)FBCheckPosReached @RT(0) @T @T @UNKNOWN 0 @F
@F @F
@T
@BEG_Attrib
3 @RT(0) @RT(0) @RT(0)
@END_Attrib
1 0 @F @F @F @F

@Var @RT(9)bMoldOpen @RT(0) @T @F @DT @RT(4)BOOL @RT(0) @T @T @BASIC 0 @F
@F @F
@T
@BEG_Attrib
3 @RT(0) @RT(0) @RT(0)
@END_Attrib
1 0 @F @F @F @F

@Var @RT(14)iImpulseActPos @RT(0) @T @F @DT @RT(4)DINT @RT(0) @T @T @BASIC 0 @F
@F @F
@T
@BEG_Attrib
3 @RT(0) @RT(54)Actual Impulse position calculated from clamping force @RT(0)
@END_Attrib
1 0 @F @F @F @F

@Var @RT(17)MovementDirection @RT(0) @T @T @DERIVED 0 @T @T @DT @RT(19)tnMovementDirection @RT(0) @T @T @UNKNOWN 0 @F
@F @F
@T
@BEG_Attrib
3 @RT(0) @RT(0) @RT(0)
@END_Attrib
1 0 @F @F @F @F

@END_Dcl

@END_Export

@BEG_SfcBody
19 12 15

@BEG_SfcData 2
@StepSeq @RT(4)sseq @F 1
@Loop @RT(4)loop @F 2
@StepSeq @RT(3)seq @F 7
@Step @RT(5)START @F @T @F @F @RT(0) @F
@AcbCont @RT(7)unnamed @F 0

@Trans @RT(10)StartTrans @F @T @F @F @T @F @TL(2)
TRUE

@RT(6)Trans1 @F
@Step @RT(16)PREPARE_MOVEMENT @F @F @F @F @RT(0) @F
@AcbCont @RT(7)unnamed @F 2
@Acb @RT(18)ACheckMoldBackward @F @F @RT(1)P @RT(0) @F @F @T @F
@Acb @RT(16)aPrepareMovement @F @F @RT(1)P @RT(0) @F @F @T @F

@AltBranch @RT(3)alt @F 3
@TransSeq @RT(4)tseq @F 1
@Trans @RT(7)TAdjust @F @T @F @F @T @F @TL(2)
bMoldOpen AND iTempImpulses <> 0

@RT(6)Trans2 @F

@TransSeq @RT(4)tseq @F 2
@Trans @RT(15)TNoAdjustNeeded @F @T @F @F @T @F @TL(2)
bMoldOpen AND iTempImpulses = 0

@RT(7)Trans13 @F
@Goto @RT(5)READY @F @F

@TransSeq @RT(4)tseq @F 2
@Trans @RT(12)TMoldNotOpen @F @T @F @F @T @F @TL(2)
NOT bMoldOpen

@RT(7)Trans14 @F
@Goto @RT(5)READY @F @F

@Step @RT(4)MOVE @F @F @F @F @RT(0) @F
@AcbCont @RT(7)unnamed @F 1
@Acb @RT(6)AReset @F @T @RT(1)P @RT(0) @F @F @T @TL(2)
sv_MoldHeightEndpoints.bPositionForStepReached := FALSE;

@F

@AltBranch @RT(3)alt @F 2
@TransSeq @RT(4)tseq @F 3
@Trans @RT(23)CheckMovementDirection1 @F @T @F @F @T @F @TL(2)
MovementDirection = nForward

@RT(6)Trans3 @F
@Step @RT(15)MOVE_FWD_TO_POS @F @F @F @F @RT(0) @F
@AcbCont @RT(7)unnamed @F 2
@Acb @RT(13)aMoveFwdToPos @F @F @RT(1)P @RT(0) @F @F @T @F
@Acb @RT(14)aCheckFwdReady @F @F @RT(1)N @RT(0) @F @F @F @F

@Trans @RT(22)CheckMovementFinished1 @F @T @F @F @T @T @TL(2)
fbCheckReady.bReady OR bStop

@RT(6)Trans5 @F

@TransSeq @RT(4)tseq @F 3
@Trans @RT(23)CheckMovementDirection2 @F @T @F @F @T @F @TL(2)
MovementDirection = nBackward

@RT(6)Trans4 @F
@Step @RT(15)MOVE_BWD_TO_POS @F @F @F @F @RT(0) @F
@AcbCont @RT(7)unnamed @F 2
@Acb @RT(13)aMoveBwdToPos @F @F @RT(1)P @RT(0) @F @F @F @F
@Acb @RT(14)aCheckBwdReady @F @F @RT(1)N @RT(0) @F @F @F @F

@Trans @RT(22)CheckMovementFinished2 @F @T @F @F @T @T @TL(2)
fbCheckReady.bReady OR bStop

@RT(6)Trans5 @F

@Step @RT(5)READY @F @F @T @F @RT(0) @F
@AcbCont @RT(7)unnamed @F 2
@Acb @RT(17)AUpdateClampForce @F @F @RT(1)P @RT(0) @F @F @T @F
@Acb @RT(18)ResetMovementFlags @F @T @RT(1)P @RT(0) @F @F @T @TL(17)
IF bStop THEN
    //stop active device
    fbStop(DeviceId := DeviceIdMoldHeight);
END_IF;

IF NOT bMoldOpen THEN
    SET_ALARM(erMoldHeightAdjustMoldNotOpen);
END_IF;

IF sv_MoldHeightEndpoints.bPositionForStepReached THEN
    SET_ALARM(erMoldHeightAdjustFinished);
ELSE
    SET_ALARM(erMoldHeightAdjustAborted);
END_IF;

bReady := TRUE;

@F

@Trans @RT(9)TLoopBack @F @T @T @T @T @T @TL(2)
TRUE

@RT(6)Trans7 @F

@END_SfcData
@SaActions 7
@SaText @RT(13)aMoveFwdToPos 1 @TL(6)
(*@ MoldHeightAdjustN.ABAdjustPositionChange.aMoveFwdToPos.Start the mold height forward movement.*)
evStartRequestData.DeviceId := DeviceIdMoldHeight;
evStartRequestData.MoveDir := cMoveFwd;
evStartRequestData.MoveId := cMoveFwd;
SET_EVENT(evStartRequest, evStartRequestData);

@SaText @RT(13)aMoveBwdToPos 1 @TL(6)
(*@ MoldHeightAdjustN.ABAdjustPositionChange.aMoveBwdToPos.Start the mold height backwar movement.*)
evStartRequestData.DeviceId := DeviceIdMoldHeight;
evStartRequestData.MoveDir := cMoveBwd;
evStartRequestData.MoveId := cMoveBwd;
SET_EVENT(evStartRequest, evStartRequestData);

@SaText @RT(16)aPrepareMovement 1 @TL(32)
(**************************************** WARNING ********************************************
 *** The KEBA Kemro K2 System including software is not intended for safety control tasks! ***
 ***                       For further information see Comment tab!                        ***
 *********************************************************************************************)

// Reset the CalcFinished and AutoAdjustFinished flag
// for normal operation.
bReady := FALSE;
iTempImpulses := 0;

abCalculateMoldHeightImpulses.aInit(Lintab := sv_ClampForceLintabImpulses);
abCalculateMoldHeightImpulses.aCalc(rForce := sv_ClampForce.rActualClampForce);
iImpulseActPos := abCalculateMoldHeightImpulses.aCalc.iImpulses;

abCalculateMoldHeightImpulses.aCalc(rForce := sv_ClampForce.rSetClampForce);
iTempImpulses := abCalculateMoldHeightImpulses.aCalc.iImpulses - iImpulseActPos;
//abCalculateMoldHeightImpulses.aCalc( rActualForce:= sv_ClampForce.rActualClampForce, rSetForce:= sv_ClampForce.rSetClampForce);
//iTempImpulses := abCalculateMoldHeightImpulses.aCalc.iImpulses;

IF iTempImpulses = 0 THEN
    bReady := TRUE;
ELSIF iTempImpulses < 0 THEN
    MovementDirection := nBackward;
    iTempImpulses := ABS(iTempImpulses);
ELSIF iTempImpulses > 0 THEN
    MovementDirection := nForward;
END_IF;

// Set the system variable for impulses to move
sv_iThisStepsSetImpulses := DINT_TO_UDINT(iTempImpulses);
sv_iThisStepsActImpulses := 0;

@SaText @RT(14)aCheckFwdReady 1 @TL(7)
(**************************************** WARNING ********************************************
 *** The KEBA Kemro K2 System including software is not intended for safety control tasks! ***
 ***                       For further information see Comment tab!                        ***
 *********************************************************************************************)

fbCheckReady(DeviceId := DeviceIdMoldHeight);

@SaText @RT(14)aCheckBwdReady 1 @TL(7)
(**************************************** WARNING ********************************************
 *** The KEBA Kemro K2 System including software is not intended for safety control tasks! ***
 ***                       For further information see Comment tab!                        ***
 *********************************************************************************************)

fbCheckReady(DeviceId := DeviceIdMoldHeight);

@SaText @RT(18)ACheckMoldBackward 1 @TL(6)

fbCheckPosReached(DeviceId := DeviceIdMold,
                  MoveDir := cMoveBwd,
                  MoveId := cMoveBwdForMHAdjust,
                  bPosReached => bMoldOpen);

@SaText @RT(17)AUpdateClampForce 1 @TL(15)
(**************************************** WARNING ********************************************
 *** The KEBA Kemro K2 System including software is not intended for safety control tasks! ***
 ***                       For further information see Comment tab!                        ***
 *********************************************************************************************)

// calculate actual new clamping foce at end of movement
abCalculateMoldHeightImpulses.aInit(Lintab := sv_ClampForceLintabImpulses);
IF MovementDirection = nForward THEN
    abCalculateMoldHeightImpulses.aCalcInv(iImpulses := iImpulseActPos + UDINT_TO_DINT(sv_iThisStepsActImpulses));
ELSE
    abCalculateMoldHeightImpulses.aCalcInv(iImpulses := iImpulseActPos - UDINT_TO_DINT(sv_iThisStepsActImpulses));
END_IF;

sv_ClampForce.rActualClampForce := abCalculateMoldHeightImpulses.aCalcInv.rForce;

@SaTrans 0
@SaExits 0
@END_SfcBody

@@@BEG_Comment@@@
@TL(5)
This algo controls the mold height automatic position change:
- A desired position is set on the hmi. By starting the automatic mold height adjustment this algo is called.
- The desired position is translated into a number of increments and direction to move to.
- The movement is started until the position reached flags are set by the movements of MoldHeight1.
- The ready flag is set and the algo won't be called any more.
@@@END_Comment@@@
@END_Body

@END_Contents

(* ---- ABAdjustPosSetTonnageDetect.pu ---- *)
(*
@h    ! WARNING !
@h    The Kemro K2 system (including software) only meets category B according to EN 954-1,
@h    thus it is not intended for usage in safety-relevant control applications in the field
@h    of personal safety (e.g. emergency stop).
@h    To implement potentially necessary safety-relevant control tasks, always use additional
@h    external safety devices that are intended for the particular purpose, and meet the necessary
@h    functional safety.
@h    For further information see EN 954-1 (EN ISO 13849-1) and/or the K2-x00 user manual, chapter
@h    "CE conformity, directives and standards".

Detect Mold Height forward end position:
Close mold
If not possible move Mold Height backward and try again
when Mold is closed move MoldHeight forward until standstill

Set clamping force:
Open mold
Move Mold Height forward by calculated number of impulses

*)

IMPORT_OVER_LISTFILE
 SET_ALARM
, REAL_TO_FORMATTED_STRING
, tevStartRequest
, KAPPL_LintabData
, tsMoldHeightPositions
, tsClampForces
, tsTraceLevel
, ABCalculateMoldHeightImpulses
, FBDebugTrace
, tsDeviceId
, FBCheckReady
, FBCheckPosReached
, tevStartRequestData
, FBStop
, ABAdjustStretchToggleLever

END_IMPORT

ALGORITHM_BLOCK ABAdjustPosSetTonnageDetect #DUMMY_EDIT_BLOCK

SYSTEM_VAR
 sv_bStandStillDetectionArmed : BOOL;
 sv_iThisStepsSetImpulses : UDINT;
 sv_ClampForceLintabImpulses : KAPPL_LintabData;
 sv_iAbsoluteImpulsesFromOrigin : DINT;
 sv_MoldHeightPositions : tsMoldHeightPositions;
 sv_ClampForce : tsClampForces;
 sv_TraceLevel : tsTraceLevel;
 sv_bOpenMHUntilProtectStep : BOOL;
END_VAR

SYSTEM_OBJECT
 evStartRequest : tevStartRequest;
 erMoldHeightAdjustAborted : ALARM;
 erMoldHeightAdjustFinished : ALARM;
END_OBJECT

VAR
 abCalculateMoldHeightImpulses : ABCalculateMoldHeightImpulses;
 fbDebugTrace : FBDebugTrace;
END_VAR

ALGORITHM aRun

VAR_INPUT
 bStop : BOOL;
END_VAR

VAR_OUTPUT
 bReady : BOOL;
END_VAR

VAR_INPUT
 DeviceIdMold : tsDeviceId;
 DeviceIdMoldHeight : tsDeviceId;
END_VAR

VAR
 bMoldOpen : BOOL;
 fbCheckReady : FBCheckReady;
 fbCheckPosReached : FBCheckPosReached;
 evStartRequestData : tevStartRequestData;
 bMoldOpenReady : BOOL;
 bMoldHeightFwdReady : BOOL;
 bFinished : BOOL;
 fbStop : FBStop;
 abAdjustStretchToggleLever : ABAdjustStretchToggleLever;
END_VAR

(* IecGraph-Code *)

(* init step *)
INITIAL_STEP START:
aPreparAdjustment (P);
END_STEP

(* steps *)
STEP S_StretchToggleLever:
aStretchToggleLever (N);
END_STEP

STEP S_CheckMoldClosed:
aCheckMoldClosed (N);
END_STEP

STEP S_MHFwdUntilStandstill:
aMoveMoldHeightFwd (P);
aCheckMoldHeightFwdReady (N);
END_STEP

STEP S_MoldOpenAfterStandstill:
aSetOrigin (P);
aOpenMold (P);
aCheckMoldOpen (N);
END_STEP

STEP S_MHFwdSetTonnage:
aMoveMoldHeightFwdSetTonnage (P);
aCheckMoldHeightFwdReady (N);
END_STEP

STEP S_CheckReady:
SetReadyFlag (P);
END_STEP

ACTION SetReadyFlag: #BEGIN_EDIT_BLOCK
bFinished := TRUE;

;#END_EDIT_BLOCK END_ACTION (*SetReadyFlag*)
STEP S_Stop:
AStop (P);
END_STEP

ACTION AStop: #BEGIN_EDIT_BLOCK
//stop active movement
IF bStop THEN
    fbStop(DeviceId := DeviceIdMold);
    fbStop(DeviceId := DeviceIdMoldHeight);
END_IF;

;#END_EDIT_BLOCK END_ACTION (*AStop*)
STEP S_Ready:
AReady (P);
END_STEP

ACTION AReady: #BEGIN_EDIT_BLOCK
IF bFinished THEN
    SET_ALARM(erMoldHeightAdjustFinished);
ELSE
    SET_ALARM(erMoldHeightAdjustAborted);
END_IF;

sv_bOpenMHUntilProtectStep := FALSE;

bReady := TRUE;

;#END_EDIT_BLOCK END_ACTION (*AReady*)

(* transitions *)
TRANSITION Trans70 FROM START TO S_StretchToggleLever :=  #BEGIN_EDIT_BLOCK
TRUE
;#END_EDIT_BLOCK
END_TRANSITION

TRANSITION TAdjustBwdReady FROM S_StretchToggleLever TO S_CheckMoldClosed :=  #BEGIN_EDIT_BLOCK
abAdjustStretchToggleLever.aRun.bReady AND
abAdjustStretchToggleLever.aRun.bSuccess
;#END_EDIT_BLOCK
END_TRANSITION

TRANSITION Trans71 FROM S_CheckMoldClosed TO S_MHFwdUntilStandstill :=  #BEGIN_EDIT_BLOCK
fbCheckReady.bReady
;#END_EDIT_BLOCK
END_TRANSITION

TRANSITION Trans72 FROM S_CheckMoldClosed TO S_Stop :=  #BEGIN_EDIT_BLOCK
NOT fbCheckReady.bReady
;#END_EDIT_BLOCK
END_TRANSITION

TRANSITION TStopAdjBwd FROM S_StretchToggleLever TO S_Stop :=  #BEGIN_EDIT_BLOCK
abAdjustStretchToggleLever.aRun.bReady AND
NOT abAdjustStretchToggleLever.aRun.bSuccess
;#END_EDIT_BLOCK
END_TRANSITION

TRANSITION TAdjFwdReady FROM S_MHFwdUntilStandstill TO S_MoldOpenAfterStandstill :=  #BEGIN_EDIT_BLOCK
bMoldHeightFwdReady
;#END_EDIT_BLOCK
END_TRANSITION

TRANSITION Trans64 FROM S_MoldOpenAfterStandstill TO S_MHFwdSetTonnage :=  #BEGIN_EDIT_BLOCK
bMoldOpenReady
// move MH forward for desired clamp force
;#END_EDIT_BLOCK
END_TRANSITION

TRANSITION TStopAdjFwd FROM S_MHFwdUntilStandstill TO S_Stop :=  #BEGIN_EDIT_BLOCK
bStop
;#END_EDIT_BLOCK
END_TRANSITION

TRANSITION Trans67 FROM S_MHFwdSetTonnage TO S_CheckReady :=  #BEGIN_EDIT_BLOCK
bMoldHeightFwdReady
;#END_EDIT_BLOCK
END_TRANSITION

TRANSITION Trans68 FROM S_MHFwdSetTonnage TO S_Stop :=  #BEGIN_EDIT_BLOCK
bStop OR (bMoldHeightFwdReady AND NOT fbCheckPosReached.bPosReached)
;#END_EDIT_BLOCK
END_TRANSITION

GO_ON_TRANSITION TFinished FROM S_CheckReady TO S_Stop :=  #BEGIN_EDIT_BLOCK
TRUE
;#END_EDIT_BLOCK
END_TRANSITION

GO_ON_TRANSITION TReady FROM S_Stop TO S_Ready :=  #BEGIN_EDIT_BLOCK
TRUE
;#END_EDIT_BLOCK
END_TRANSITION

TRANSITION Trans33 FROM S_Ready TO START :=  #BEGIN_EDIT_BLOCK
TRUE
;#END_EDIT_BLOCK
END_TRANSITION

(* end IecGraph-Code *)
(* sfc-code *)

(* stand alone actions *)
ACTION aPreparAdjustment: #BEGIN_EDIT_BLOCK
bReady := FALSE;
bFinished := FALSE;

IF sv_TraceLevel.bApplication THEN
    fbDebugTrace(sText := 'MoldHeightAuto: start');
END_IF;

;#END_EDIT_BLOCK END_ACTION (*aPreparAdjustment*)
ACTION aOpenMold: #BEGIN_EDIT_BLOCK
// Start the mold open movement until protect step
IF sv_TraceLevel.bApplication THEN
    fbDebugTrace(sText := 'MoldHeightAuto: opening Mold');
END_IF;

sv_bOpenMHUntilProtectStep := TRUE;

evStartRequestData.DeviceId := DeviceIdMold;
evStartRequestData.MoveDir := cMoveBwd;
evStartRequestData.MoveId := cMoveBwdForMHAdjustSetup;
SET_EVENT(evStartRequest, evStartRequestData);

;#END_EDIT_BLOCK END_ACTION (*aOpenMold*)
ACTION aMoveMoldHeightFwd: #BEGIN_EDIT_BLOCK
(*@ MoldHeightAdjustN.ABAdjustForceOpenLoop.paRun.aMoveMoldHeightFwd.Because the mold height forward movement
                                                    can be stopped by either the detection of a stand still or
                                                    the reaching of desired impulses for this step, these two
                                                    conditions are combined into the bMoldHeightFwdReady flag.
                                                    Of course this flag has to be reset when the movement starts*)

IF sv_TraceLevel.bApplication THEN
    fbDebugTrace(sText := 'MoldHeightAuto: MH forward until standstill');
END_IF;

bMoldHeightFwdReady := FALSE;
sv_bStandStillDetectionArmed := TRUE;
sv_iThisStepsSetImpulses := 100000;

// Start the mold height forward movement
evStartRequestData.DeviceId := DeviceIdMoldHeight;
evStartRequestData.MoveDir := cMoveFwd;
evStartRequestData.MoveId := cMoveFwd;
SET_EVENT(evStartRequest, evStartRequestData);

;#END_EDIT_BLOCK END_ACTION (*aMoveMoldHeightFwd*)
ACTION aCheckMoldHeightFwdReady: #BEGIN_EDIT_BLOCK
(**************************************** WARNING ********************************************
 *** The KEBA Kemro K2 System including software is not intended for safety control tasks! ***
 ***                       For further information see Comment tab!                        ***
 *********************************************************************************************)

fbCheckReady(DeviceId := DeviceIdMoldHeight,
             bReady => bMoldHeightFwdReady);

fbCheckPosReached(DeviceId := DeviceIdMoldHeight,
                  MoveDir := cMoveFwd,
                  MoveId := cMoveFwd(*,
                  bPosReached => *));

;#END_EDIT_BLOCK END_ACTION (*aCheckMoldHeightFwdReady*)
ACTION aCheckMoldOpen: #BEGIN_EDIT_BLOCK
(*@ MoldHeightAdjustN.ABAdjustForceOpenLoop.paRun.aCheckMoldOpen.Check the status of mold open movement
                                                    - Finished
                                                    - PositionReached*)
fbCheckReady(DeviceId := DeviceIdMold,
             bReady => bMoldOpenReady);
fbCheckPosReached(DeviceId := DeviceIdMold,
                  MoveDir := cMoveBwd,
                  MoveId := cMoveBwdForMHAdjustSetup,
                  bPosReached => bMoldOpen);

;#END_EDIT_BLOCK END_ACTION (*aCheckMoldOpen*)
ACTION aMoveMoldHeightFwdSetTonnage: #BEGIN_EDIT_BLOCK

sv_ClampForce.rActualClampForce := sv_ClampForce.rSetClampForce;
abCalculateMoldHeightImpulses.aInit(Lintab := sv_ClampForceLintabImpulses);
abCalculateMoldHeightImpulses.aCalc(rForce:=sv_ClampForce.rSetClampForce);

//enable standstill detection in case we want to move too far
sv_bStandStillDetectionArmed := TRUE;
sv_iThisStepsSetImpulses := DINT_TO_UDINT(abCalculateMoldHeightImpulses.aCalc.iImpulses);

IF sv_TraceLevel.bApplication THEN
    fbDebugTrace(sText := CONCAT('MoldHeightAuto: MH forward for setting clamp force ',
                                 REAL_TO_FORMATTED_STRING(sv_ClampForce.rSetClampForce, 4, 1),' -->',
                                 UDINT_TO_STRING(sv_iThisStepsSetImpulses)));
END_IF;

// Start the mold height forward movement
evStartRequestData.DeviceId := DeviceIdMoldHeight;
evStartRequestData.MoveDir := cMoveFwd;
evStartRequestData.MoveId := cMoveFwd;
SET_EVENT(evStartRequest, evStartRequestData);

;#END_EDIT_BLOCK END_ACTION (*aMoveMoldHeightFwdSetTonnage*)
ACTION aSetOrigin: #BEGIN_EDIT_BLOCK

IF sv_TraceLevel.bApplication THEN

    fbDebugTrace(sText := CONCAT('MoldHeightAuto: setting new origin, old one at',DINT_TO_STRING(sv_iAbsoluteImpulsesFromOrigin)));
END_IF;

// we are at the mold height origin = 0 impulses away from 0.0 mm
sv_iAbsoluteImpulsesFromOrigin := 0;
sv_MoldHeightPositions.rOriginMoldHeightPosition := 0.0;

//sv_MoldHeightPositions.rMaxMoldHeightPosition := ? needed?
//sv_MoldHeightPositions.rMinMoldHeightPosition := ? needed?
//sv_MoldHeightPositions.rMoveToMoldHeightPosition := ?

;#END_EDIT_BLOCK END_ACTION (*aSetOrigin*)
ACTION aStretchToggleLever: #BEGIN_EDIT_BLOCK
abAdjustStretchToggleLever.aRun(bStop := bStop, DeviceIdMold := DeviceIdMold,
                                DeviceIdMoldHeight := DeviceIdMoldHeight,
                                bUseImpulses := TRUE, iImpulses := 64);

;#END_EDIT_BLOCK END_ACTION (*aStretchToggleLever*)
ACTION aCheckMoldClosed: #BEGIN_EDIT_BLOCK
//Check the status of mold close movement
// - Finished
// - PositionReached
fbCheckReady(DeviceId := DeviceIdMold);
fbCheckPosReached(DeviceId := DeviceIdMold,
                  MoveDir := cMoveFwd,
                  MoveId := cMoveFwdForMHAdjustSetup);

;#END_EDIT_BLOCK END_ACTION (*aCheckMoldClosed*)
(* end sfc-code *)

END_ALGORITHM

END_ALGORITHM_BLOCK

#END_OF_IEC_PART

@Puma @IecEditor 6 30 @Pou 25
@@@BEG_Comment@@@
@h    ! WARNING !
@h    The Kemro K2 system (including software) only meets category B according to EN 954-1,
@h    thus it is not intended for usage in safety-relevant control applications in the field
@h    of personal safety (e.g. emergency stop).
@h    To implement potentially necessary safety-relevant control tasks, always use additional
@h    external safety devices that are intended for the particular purpose, and meet the necessary
@h    functional safety.
@h    For further information see EN 954-1 (EN ISO 13849-1) and/or the K2-x00 user manual, chapter
@h    "CE conformity, directives and standards".

Detect Mold Height forward end position:
Close mold
If not possible move Mold Height backward and try again
when Mold is closed move MoldHeight forward until standstill

Set clamping force:
Open mold
Move Mold Height forward by calculated number of impulses

@@@END_Comment@@@

@BEG_Contents

@BEG_Func
@RT(17)FuncTreeContainer
2
@Var @RT(9)SET_ALARM @RT(0) @T @T @DERIVED 0 @F @RT(23)KEBA_STANDARD_PROCEDURE @F
@T
@BEG_Attrib
0 @RT(0) @RT(0)
@END_Attrib
1 1 @F @F @F @F

@Var @RT(24)REAL_TO_FORMATTED_STRING @RT(0) @T @T @DERIVED 0 @F @RT(22)KEBA_STANDARD_FUNCTION @F
@T
@BEG_Attrib
0 @RT(0) @RT(0)
@END_Attrib
1 1 @F @F @F @F

@END_Func

@BEG_Const
@RT(18)ConstTreeContainer
0
@END_Const

@BEG_Export

@BEG_Kind
@ALGORITHM_BLOCK @RT(27)ABAdjustPosSetTonnageDetect @STRUCTURED_TEXT
@RT(0) @RT(0) @RT(0)
@END_Kind

@BEG_Dcl
@RT(16)DclTreeContainer
13
@Var @RT(14)evStartRequest @RT(0) @T @T @DERIVED 0 @T @T @DT @RT(15)tevStartRequest @RT(0) @T @T @UNKNOWN 0 @F
@F @F
@T
@BEG_Attrib
3 @RT(0) @RT(0) @RT(0)
@END_Attrib
1 7 @F @F @F @F

@Var @RT(25)erMoldHeightAdjustAborted @RT(0) @T @F @DT @RT(5)ALARM @RT(0) @T @T @BASIC 0 @F
@F @F
@T
@BEG_Attrib
3 @RT(0) @RT(0) @RT(0)
@END_Attrib
1 7 @F @F @F @F

@Var @RT(26)erMoldHeightAdjustFinished @RT(0) @T @F @DT @RT(5)ALARM @RT(0) @T @T @BASIC 0 @F
@F @F
@T
@BEG_Attrib
3 @RT(0) @RT(0) @RT(0)
@END_Attrib
1 7 @F @F @F @F

@Var @RT(28)sv_bStandStillDetectionArmed @RT(0) @T @T @RENAMED 0 @T @T @DT @RT(4)BOOL @RT(0) @T @T @BASIC 0 @F
@F @F
@T
@BEG_Attrib
3 @RT(0) @RT(0) @RT(0)
@END_Attrib
1 8 @F @F @F @F

@Var @RT(24)sv_iThisStepsSetImpulses @RT(0) @T @F @DT @RT(5)UDINT @RT(0) @T @T @BASIC 0 @F
@F @F
@T
@BEG_Attrib
3 @RT(0) @RT(0) @RT(0)
@END_Attrib
1 8 @F @F @F @F

@Var @RT(27)sv_ClampForceLintabImpulses @RT(0) @T @T @DERIVED 0 @T @T @DT @RT(16)KAPPL_LintabData @RT(0) @T @T @UNKNOWN 0 @F
@F @F
@T
@BEG_Attrib
3 @RT(0) @RT(0) @RT(0)
@END_Attrib
1 8 @F @F @F @F

@Var @RT(30)sv_iAbsoluteImpulsesFromOrigin @RT(0) @T @T @RENAMED 0 @T @T @DT @RT(4)DINT @RT(0) @T @T @BASIC 0 @F
@F @F
@T
@BEG_Attrib
3 @RT(0) @RT(0) @RT(0)
@END_Attrib
1 8 @F @F @F @F

@Var @RT(22)sv_MoldHeightPositions @RT(0) @T @T @DERIVED 0 @T @T @DT @RT(21)tsMoldHeightPositions @RT(0) @T @T @UNKNOWN 0 @F
@F @F
@T
@BEG_Attrib
3 @RT(0) @RT(0) @RT(0)
@END_Attrib
1 8 @F @F @F @F

@Var @RT(13)sv_ClampForce @RT(0) @T @T @DERIVED 0 @T @T @DT @RT(13)tsClampForces @RT(0) @T @T @UNKNOWN 0 @F
@F @F
@T
@BEG_Attrib
3 @RT(0) @RT(0) @RT(0)
@END_Attrib
1 8 @F @F @F @F

@Var @RT(13)sv_TraceLevel @RT(0) @T @T @RENAMED 0 @T @T @DT @RT(12)tsTraceLevel @RT(0) @T @T @UNKNOWN 0 @F
@F @F
@T
@BEG_Attrib
3 @RT(0) @RT(0) @RT(0)
@END_Attrib
1 8 @F @F @F @F

@Var @RT(29)abCalculateMoldHeightImpulses @RT(0) @T @T @DERIVED 0 @T @T @DT @RT(29)ABCalculateMoldHeightImpulses @RT(0) @T @T @UNKNOWN 0 @F
@F @F
@T
@BEG_Attrib
3 @RT(0) @RT(0) @RT(0)
@END_Attrib
1 0 @F @F @F @F

@Var @RT(12)fbDebugTrace @RT(0) @T @T @DERIVED 0 @T @T @DT @RT(12)FBDebugTrace @RT(0) @T @T @UNKNOWN 0 @F
@F @F
@T
@BEG_Attrib
3 @RT(0) @RT(0) @RT(0)
@END_Attrib
1 0 @F @F @F @F

@Var @RT(26)sv_bOpenMHUntilProtectStep @RT(0) @T @T @RENAMED 0 @T @T @DT @RT(4)BOOL @RT(0) @T @T @BASIC 0 @F
@F @F
@T
@BEG_Attrib
3 @RT(0) @RT(0) @RT(0)
@END_Attrib
1 8 @F @F @F @F

@END_Dcl

@END_Export

@BEG_Body

1

@BEG_Export

@BEG_Algo
@ALGORITHM @RT(4)aRun @SEQUENTIAL_FLOW_CHART
@RT(0) @RT(0) @RT(0) @F @F
@END_Algo

@BEG_Dcl
@RT(16)DclTreeContainer
13
@Var @RT(5)bStop @RT(0) @T @F @DT @RT(4)BOOL @RT(0) @T @T @BASIC 0 @F
@F @F
@T
@BEG_Attrib
3 @RT(0) @RT(0) @RT(0)
@END_Attrib
1 1 @F @F @F @F

@Var @RT(6)bReady @RT(0) @T @F @DT @RT(4)BOOL @RT(0) @T @T @BASIC 0 @F
@F @F
@T
@BEG_Attrib
3 @RT(0) @RT(0) @RT(0)
@END_Attrib
1 3 @F @F @F @F

@Var @RT(12)DeviceIdMold @RT(0) @T @T @DERIVED 0 @T @T @DT @RT(10)tsDeviceId @RT(0) @T @T @UNKNOWN 0 @F
@F @F
@T
@BEG_Attrib
3 @RT(0) @RT(0) @RT(0)
@END_Attrib
1 1 @F @F @F @F

@Var @RT(18)DeviceIdMoldHeight @RT(0) @T @T @DERIVED 0 @T @T @DT @RT(10)tsDeviceId @RT(0) @T @T @UNKNOWN 0 @F
@F @F
@T
@BEG_Attrib
3 @RT(0) @RT(0) @RT(0)
@END_Attrib
1 1 @F @F @F @F

@Var @RT(9)bMoldOpen @RT(0) @T @F @DT @RT(4)BOOL @RT(0) @T @T @BASIC 0 @F
@F @F
@T
@BEG_Attrib
3 @RT(0) @RT(0) @RT(0)
@END_Attrib
1 0 @F @F @F @F

@Var @RT(12)fbCheckReady @RT(0) @T @T @DERIVED 0 @T @T @DT @RT(12)FBCheckReady @RT(0) @T @T @UNKNOWN 0 @F
@F @F
@T
@BEG_Attrib
3 @RT(0) @RT(0) @RT(0)
@END_Attrib
1 0 @F @F @F @F

@Var @RT(17)fbCheckPosReached @RT(0) @T @T @DERIVED 0 @T @T @DT @RT(17)FBCheckPosReached @RT(0) @T @T @UNKNOWN 0 @F
@F @F
@T
@BEG_Attrib
3 @RT(0) @RT(0) @RT(0)
@END_Attrib
1 0 @F @F @F @F

@Var @RT(18)evStartRequestData @RT(0) @T @T @DERIVED 0 @T @T @DT @RT(19)tevStartRequestData @RT(0) @T @T @UNKNOWN 0 @F
@F @F
@T
@BEG_Attrib
3 @RT(0) @RT(0) @RT(0)
@END_Attrib
1 0 @F @F @F @F

@Var @RT(14)bMoldOpenReady @RT(0) @T @F @DT @RT(4)BOOL @RT(0) @T @T @BASIC 0 @F
@F @F
@T
@BEG_Attrib
3 @RT(0) @RT(0) @RT(0)
@END_Attrib
1 0 @F @F @F @F

@Var @RT(19)bMoldHeightFwdReady @RT(0) @T @F @DT @RT(4)BOOL @RT(0) @T @T @BASIC 0 @F
@F @F
@T
@BEG_Attrib
3 @RT(0) @RT(0) @RT(0)
@END_Attrib
1 0 @F @F @F @F

@Var @RT(9)bFinished @RT(0) @T @F @DT @RT(4)BOOL @RT(0) @T @T @BASIC 0 @F
@F @F
@T
@BEG_Attrib
3 @RT(0) @RT(0) @RT(0)
@END_Attrib
1 0 @F @F @F @F

@Var @RT(6)fbStop @RT(0) @T @T @DERIVED 0 @T @T @DT @RT(6)FBStop @RT(0) @T @T @UNKNOWN 0 @F
@F @F
@T
@BEG_Attrib
3 @RT(0) @RT(0) @RT(0)
@END_Attrib
1 0 @F @F @F @F

@Var @RT(26)abAdjustStretchToggleLever @RT(0) @T @T @DERIVED 0 @T @T @DT @RT(26)ABAdjustStretchToggleLever @RT(0) @T @T @UNKNOWN 0 @F
@F @F
@T
@BEG_Attrib
3 @RT(0) @RT(0) @RT(0)
@END_Attrib
1 0 @F @F @F @F

@END_Dcl

@END_Export

@BEG_SfcBody
62 47 73

@BEG_SfcData 2
@StepSeq @RT(4)sseq @F 1
@Loop @RT(4)loop @F 2
@StepSeq @RT(3)seq @F 13
@Step @RT(5)START @F @T @F @F @RT(0) @F
@AcbCont @RT(7)unnamed @F 1
@Acb @RT(17)aPreparAdjustment @F @F @RT(1)P @RT(0) @F @F @T @F

@Trans @RT(7)Trans70 @F @T @F @F @T @T @TL(2)
TRUE

@RT(7)Trans70 @F
@Step @RT(20)S_StretchToggleLever @F @F @F @F @RT(0) @F
@AcbCont @RT(7)unnamed @F 1
@Acb @RT(19)aStretchToggleLever @F @F @RT(1)N @RT(0) @F @F @T @F

@AltBranch @RT(3)alt @F 2
@TransSeq @RT(4)tseq @F 3
@Trans @RT(15)TAdjustBwdReady @F @T @F @F @T @T @TL(3)
abAdjustStretchToggleLever.aRun.bReady AND
abAdjustStretchToggleLever.aRun.bSuccess

@RT(7)Trans38 @F
@Step @RT(17)S_CheckMoldClosed @F @F @F @F @RT(0) @F
@AcbCont @RT(7)unnamed @F 1
@Acb @RT(16)aCheckMoldClosed @F @F @RT(1)N @RT(0) @F @F @T @T @TL(1)
Comment :be paranoid and check if really closed

@AltBranch @RT(3)alt @F 2
@TransSeq @RT(4)tseq @F 1
@Trans @RT(7)Trans71 @F @T @F @F @T @T @TL(2)
fbCheckReady.bReady

@RT(7)Trans71 @F

@TransSeq @RT(4)tseq @F 2
@Trans @RT(7)Trans72 @F @T @F @F @T @T @TL(2)
NOT fbCheckReady.bReady

@RT(7)Trans72 @F
@Goto @RT(6)S_Stop @F @F

@TransSeq @RT(4)tseq @F 2
@Trans @RT(11)TStopAdjBwd @F @T @F @F @T @T @TL(3)
abAdjustStretchToggleLever.aRun.bReady AND
NOT abAdjustStretchToggleLever.aRun.bSuccess

@RT(7)Trans39 @F
@Goto @RT(6)S_Stop @F @F

@Step @RT(22)S_MHFwdUntilStandstill @F @F @F @F @RT(0) @F
@AcbCont @RT(7)unnamed @F 2
@Acb @RT(18)aMoveMoldHeightFwd @F @F @RT(1)P @RT(0) @F @F @T @F
@Acb @RT(24)aCheckMoldHeightFwdReady @F @F @RT(1)N @RT(0) @F @F @T @F

@AltBranch @RT(3)alt @F 2
@TransSeq @RT(4)tseq @F 3
@Trans @RT(12)TAdjFwdReady @F @T @F @F @T @T @TL(2)
bMoldHeightFwdReady

@RT(7)Trans41 @F
@Step @RT(25)S_MoldOpenAfterStandstill @F @F @F @F @RT(0) @F
@AcbCont @RT(7)unnamed @F 3
@Acb @RT(10)aSetOrigin @F @F @RT(1)P @RT(0) @F @F @T @F
@Acb @RT(9)aOpenMold @F @F @RT(1)P @RT(0) @F @F @T @F
@Acb @RT(14)aCheckMoldOpen @F @F @RT(1)N @RT(0) @F @F @T @F

@Trans @RT(7)Trans64 @F @T @F @F @T @T @TL(3)
bMoldOpenReady
// move MH forward for desired clamp force

@RT(7)Trans64 @F

@TransSeq @RT(4)tseq @F 2
@Trans @RT(11)TStopAdjFwd @F @T @F @F @T @T @TL(2)
bStop

@RT(7)Trans42 @F
@Goto @RT(6)S_Stop @F @F

@Step @RT(17)S_MHFwdSetTonnage @F @F @F @F @RT(0) @F
@AcbCont @RT(7)unnamed @F 2
@Acb @RT(28)aMoveMoldHeightFwdSetTonnage @F @F @RT(1)P @RT(0) @F @F @T @F
@Acb @RT(24)aCheckMoldHeightFwdReady @F @F @RT(1)N @RT(0) @F @F @T @F

@AltBranch @RT(3)alt @F 2
@TransSeq @RT(4)tseq @F 1
@Trans @RT(7)Trans67 @F @T @F @F @T @T @TL(2)
bMoldHeightFwdReady

@RT(7)Trans67 @F

@TransSeq @RT(4)tseq @F 2
@Trans @RT(7)Trans68 @F @T @F @F @T @T @TL(2)
bStop OR (bMoldHeightFwdReady AND NOT fbCheckPosReached.bPosReached)

@RT(7)Trans68 @F
@Goto @RT(6)S_Stop @F @F

@Step @RT(12)S_CheckReady @F @F @F @F @RT(0) @F
@AcbCont @RT(7)unnamed @F 1
@Acb @RT(12)SetReadyFlag @F @T @RT(1)P @RT(0) @F @F @T @TL(2)
bFinished := TRUE;

@F

@Trans @RT(9)TFinished @F @T @F @F @T @F @TL(2)
TRUE

@RT(7)Trans30 @F
@Step @RT(6)S_Stop @F @F @T @F @RT(0) @F
@AcbCont @RT(7)unnamed @F 1
@Acb @RT(5)AStop @F @T @RT(1)P @RT(0) @F @F @T @TL(6)
//stop active movement
IF bStop THEN
    fbStop(DeviceId := DeviceIdMold);
    fbStop(DeviceId := DeviceIdMoldHeight);
END_IF;

@F

@Trans @RT(6)TReady @F @T @F @F @T @F @TL(2)
TRUE

@RT(7)Trans32 @F
@Step @RT(7)S_Ready @F @F @F @F @RT(0) @F
@AcbCont @RT(7)unnamed @F 1
@Acb @RT(6)AReady @F @T @RT(1)P @RT(0) @F @F @T @TL(10)
IF bFinished THEN
    SET_ALARM(erMoldHeightAdjustFinished);
ELSE
    SET_ALARM(erMoldHeightAdjustAborted);
END_IF;

sv_bOpenMHUntilProtectStep := FALSE;

bReady := TRUE;

@F

@Trans @RT(7)Trans33 @F @T @T @T @T @T @TL(2)
TRUE

@RT(7)Trans33 @F

@END_SfcData
@SaActions 9
@SaText @RT(17)aPreparAdjustment 1 @TL(8)
bReady := FALSE;
bFinished := FALSE;

IF sv_TraceLevel.bApplication THEN
    fbDebugTrace(sText := 'MoldHeightAuto: start');
END_IF;

@SaText @RT(9)aOpenMold 1 @TL(12)
// Start the mold open movement until protect step
IF sv_TraceLevel.bApplication THEN
    fbDebugTrace(sText := 'MoldHeightAuto: opening Mold');
END_IF;

sv_bOpenMHUntilProtectStep := TRUE;

evStartRequestData.DeviceId := DeviceIdMold;
evStartRequestData.MoveDir := cMoveBwd;
evStartRequestData.MoveId := cMoveBwdForMHAdjustSetup;
SET_EVENT(evStartRequest, evStartRequestData);

@SaText @RT(18)aMoveMoldHeightFwd 1 @TL(23)
(*@ MoldHeightAdjustN.ABAdjustForceOpenLoop.paRun.aMoveMoldHeightFwd.Because the mold height forward movement
                                                    can be stopped by either the detection of a stand still or
                                                    the reaching of desired impulses for this step, these two
                                                    conditions are combined into the bMoldHeightFwdReady flag.
                                                    Of course this flag has to be reset when the movement starts*)

IF sv_TraceLevel.bApplication THEN
    fbDebugTrace(sText := 'MoldHeightAuto: MH forward until standstill');
END_IF;

bMoldHeightFwdReady := FALSE;
sv_bStandStillDetectionArmed := TRUE;
sv_iThisStepsSetImpulses := 100000;

// Start the mold height forward movement
evStartRequestData.DeviceId := DeviceIdMoldHeight;
evStartRequestData.MoveDir := cMoveFwd;
evStartRequestData.MoveId := cMoveFwd;
SET_EVENT(evStartRequest, evStartRequestData);

@SaText @RT(24)aCheckMoldHeightFwdReady 1 @TL(13)
(**************************************** WARNING ********************************************
 *** The KEBA Kemro K2 System including software is not intended for safety control tasks! ***
 ***                       For further information see Comment tab!                        ***
 *********************************************************************************************)

fbCheckReady(DeviceId := DeviceIdMoldHeight,
             bReady => bMoldHeightFwdReady);

fbCheckPosReached(DeviceId := DeviceIdMoldHeight,
                  MoveDir := cMoveFwd,
                  MoveId := cMoveFwd(*,
                  bPosReached => *));

@SaText @RT(14)aCheckMoldOpen 1 @TL(10)
(*@ MoldHeightAdjustN.ABAdjustForceOpenLoop.paRun.aCheckMoldOpen.Check the status of mold open movement
                                                    - Finished
                                                    - PositionReached*)
fbCheckReady(DeviceId := DeviceIdMold,
             bReady => bMoldOpenReady);
fbCheckPosReached(DeviceId := DeviceIdMold,
                  MoveDir := cMoveBwd,
                  MoveId := cMoveBwdForMHAdjustSetup,
                  bPosReached => bMoldOpen);

@SaText @RT(28)aMoveMoldHeightFwdSetTonnage 1 @TL(22)

sv_ClampForce.rActualClampForce := sv_ClampForce.rSetClampForce;
abCalculateMoldHeightImpulses.aInit(Lintab := sv_ClampForceLintabImpulses);
abCalculateMoldHeightImpulses.aCalc(rForce:=sv_ClampForce.rSetClampForce);

//enable standstill detection in case we want to move too far
sv_bStandStillDetectionArmed := TRUE;
sv_iThisStepsSetImpulses := DINT_TO_UDINT(abCalculateMoldHeightImpulses.aCalc.iImpulses);

IF sv_TraceLevel.bApplication THEN
    fbDebugTrace(sText := CONCAT('MoldHeightAuto: MH forward for setting clamp force ',
                                 REAL_TO_FORMATTED_STRING(sv_ClampForce.rSetClampForce, 4, 1),' -->',
                                 UDINT_TO_STRING(sv_iThisStepsSetImpulses)));
END_IF;

// Start the mold height forward movement
evStartRequestData.DeviceId := DeviceIdMoldHeight;
evStartRequestData.MoveDir := cMoveFwd;
evStartRequestData.MoveId := cMoveFwd;
SET_EVENT(evStartRequest, evStartRequestData);

@SaText @RT(10)aSetOrigin 1 @TL(14)

IF sv_TraceLevel.bApplication THEN

    fbDebugTrace(sText := CONCAT('MoldHeightAuto: setting new origin, old one at',DINT_TO_STRING(sv_iAbsoluteImpulsesFromOrigin)));
END_IF;

// we are at the mold height origin = 0 impulses away from 0.0 mm
sv_iAbsoluteImpulsesFromOrigin := 0;
sv_MoldHeightPositions.rOriginMoldHeightPosition := 0.0;

//sv_MoldHeightPositions.rMaxMoldHeightPosition := ? needed?
//sv_MoldHeightPositions.rMinMoldHeightPosition := ? needed?
//sv_MoldHeightPositions.rMoveToMoldHeightPosition := ?

@SaText @RT(19)aStretchToggleLever 1 @TL(4)
abAdjustStretchToggleLever.aRun(bStop := bStop, DeviceIdMold := DeviceIdMold,
                                DeviceIdMoldHeight := DeviceIdMoldHeight,
                                bUseImpulses := TRUE, iImpulses := 64);

@SaText @RT(16)aCheckMoldClosed 1 @TL(8)
//Check the status of mold close movement
// - Finished
// - PositionReached
fbCheckReady(DeviceId := DeviceIdMold);
fbCheckPosReached(DeviceId := DeviceIdMold,
                  MoveDir := cMoveFwd,
                  MoveId := cMoveFwdForMHAdjustSetup);

@SaTrans 0
@SaExits 0
@END_SfcBody

@@@BEG_Comment@@@
@TL(0)

@@@END_Comment@@@
@END_Body

@END_Contents

(* ---- ABAdjustStretchToggleLever.pu ---- *)
(*
@h    ! WARNING !
@h    The Kemro K2 system (including software) only meets category B according to EN 954-1,
@h    thus it is not intended for usage in safety-relevant control applications in the field
@h    of personal safety (e.g. emergency stop).
@h    To implement potentially necessary safety-relevant control tasks, always use additional
@h    external safety devices that are intended for the particular purpose, and meet the necessary
@h    functional safety.
@h    For further information see EN 954-1 (EN ISO 13849-1) and/or the K2-x00 user manual, chapter
@h    "CE conformity, directives and standards".

Helper for mold height adjustment
try to stretch the toggle lever
if not possible move backward a defined pos
*)

IMPORT_OVER_LISTFILE
 SET_ALARM
, REAL_TO_FORMATTED_STRING
, tevStartRequest
, tsTraceLevel
, FBDebugTrace
, tsDeviceId
, FBCheckReady
, FBCheckPosReached
, tevStartRequestData
, FBStop
, FBMoveMHTimeOrImpulses

END_IMPORT

ALGORITHM_BLOCK ABAdjustStretchToggleLever #DUMMY_EDIT_BLOCK

SYSTEM_VAR
 sv_TraceLevel : tsTraceLevel;
 sv_bOpenMHUntilProtectStep : BOOL;
END_VAR

SYSTEM_OBJECT
 evStartRequest : tevStartRequest;
 erMoldHeightAdjustAborted : ALARM;
END_OBJECT

VAR
 fbDebugTrace : FBDebugTrace;
END_VAR

(*
Stretch the toggle lever:

try to close mold
if not possible (standstill before pos 0)
  open mold again
  move mold height backward
  try again

mold close possible -> done
*)

ALGORITHM aRun

VAR_INPUT
 bStop : BOOL;
 DeviceIdMold : tsDeviceId;
 DeviceIdMoldHeight : tsDeviceId;
 bUseImpulses : BOOL (* TRUE: count impulses in bwd movement FALSE: timed bwd movement *);
 iImpulses : UDINT (* impulses to move backward if mold can not close *);
 dTime : TIME (* time to move backward if mold can not close *);
END_VAR

VAR_OUTPUT
 bReady : BOOL (* movement stopped with error or success *);
 bSuccess : BOOL (* if the toggle lever could be stretched *);
END_VAR

VAR
 bMoldOpen : BOOL;
 fbCheckReady : FBCheckReady;
 fbCheckPosReached : FBCheckPosReached;
 evStartRequestData : tevStartRequestData;
 bMoldClosed : BOOL;
 bMoldCloseReady : BOOL;
 bMoldOpenReady : BOOL;
 fbStop : FBStop;
 dWaitAfterCloseDelay : TIME := t#100ms;
 fbMoveTimeOrImpulses : FBMoveMHTimeOrImpulses;
END_VAR

(* IecGraph-Code *)

(* init step *)
INITIAL_STEP START:
aPreparAdjustment (P);
END_STEP

(* steps *)
STEP S_MoldClose:
aCloseMold (P);
aCheckMoldClosed (N);
END_STEP

STEP Step35:
END_STEP

STEP S_OpenMold:
aOpenMold (P);
aCheckMoldOpen (N);
END_STEP

STEP S_MHBwd:
Action66 (N);
END_STEP

ACTION Action66: #BEGIN_EDIT_BLOCK
fbMoveTimeOrImpulses(bUseImpulses := bUseImpulses, dTime := dTime, iImpulses := iImpulses,
                    DeviceId := DeviceIdMoldHeight, MoveDir := cMoveBwd, MoveId := cMoveBwd);

;#END_EDIT_BLOCK END_ACTION (*Action66*)
STEP Step26:
END_STEP

STEP Step50:
Action67 (N);
END_STEP

ACTION Action67: #BEGIN_EDIT_BLOCK
SET_ALARM(erMoldHeightAdjustAborted);
//FIXME: maybe use different alarm

;#END_EDIT_BLOCK END_ACTION (*Action67*)
STEP S_TryAgain:
END_STEP

STEP S_Done:
aDone (P);
END_STEP

ACTION aDone: #BEGIN_EDIT_BLOCK
//toggle lever is stretched
bSuccess := TRUE;

;#END_EDIT_BLOCK END_ACTION (*aDone*)
STEP S_Stop:
aFailed (N);
END_STEP

ACTION aFailed: #BEGIN_EDIT_BLOCK
bSuccess := FALSE;

;#END_EDIT_BLOCK END_ACTION (*aFailed*)
STEP S_Restart:
AStop (P);
END_STEP

ACTION AStop: #BEGIN_EDIT_BLOCK
//stop active movement
IF bStop THEN
    fbStop(DeviceId := DeviceIdMold);
    fbStop(DeviceId := DeviceIdMoldHeight);
END_IF;

sv_bOpenMHUntilProtectStep :=FALSE;

bReady := TRUE;

;#END_EDIT_BLOCK END_ACTION (*AStop*)

(* transitions *)
TRANSITION TStart FROM START TO S_MoldClose :=  #BEGIN_EDIT_BLOCK
TRUE
;#END_EDIT_BLOCK
END_TRANSITION

TRANSITION TMoldCloseReady FROM S_MoldClose TO Step35 :=  #BEGIN_EDIT_BLOCK
S_MoldClose.T >= dWaitAfterCloseDelay AND bMoldCloseReady
;#END_EDIT_BLOCK
END_TRANSITION

GO_ON_TRANSITION Trans54 FROM Step35 TO S_OpenMold :=  #BEGIN_EDIT_BLOCK
NOT bMoldClosed
;#END_EDIT_BLOCK
END_TRANSITION

GO_ON_TRANSITION TMoldClosed FROM Step35 TO S_Done :=  #BEGIN_EDIT_BLOCK
bMoldClosed
// mold could be closed,
// our part is done
;#END_EDIT_BLOCK
END_TRANSITION

TRANSITION TStopMoldClose FROM S_MoldClose TO S_Stop :=  #BEGIN_EDIT_BLOCK
S_MoldClose.T >= dWaitAfterCloseDelay AND bStop
;#END_EDIT_BLOCK
END_TRANSITION

TRANSITION TMoldIsOpen FROM S_OpenMold TO S_MHBwd :=  #BEGIN_EDIT_BLOCK
bMoldOpenReady
;#END_EDIT_BLOCK
END_TRANSITION

TRANSITION Trans76 FROM S_OpenMold TO S_Stop :=  #BEGIN_EDIT_BLOCK
bStop
;#END_EDIT_BLOCK
END_TRANSITION

TRANSITION TAdjustBwdReady FROM S_MHBwd TO Step26 :=  #BEGIN_EDIT_BLOCK
fbMoveTimeOrImpulses.bDone

//AND
//fbMoveTimeOrImpulses.
//bAdjustBwdReady
;#END_EDIT_BLOCK
END_TRANSITION

TRANSITION TStopAdjBwd FROM S_MHBwd TO S_Stop :=  #BEGIN_EDIT_BLOCK
bStop

//OR
//(fbMoveTimeOrImpulses.bDone AND NOT fbMoveTimeOrImpulses.bAtTargetPos)
;#END_EDIT_BLOCK
END_TRANSITION

GO_ON_TRANSITION AdjBwdPosReached FROM Step26 TO S_TryAgain :=  #BEGIN_EDIT_BLOCK
fbMoveTimeOrImpulses.bAtTargetPos

//sv_MoldHeightEndpoints.bPositionForStepReached
;#END_EDIT_BLOCK
END_TRANSITION

GO_ON_TRANSITION AdjBwdPosNotReached FROM Step26 TO Step50 :=  #BEGIN_EDIT_BLOCK
NOT fbMoveTimeOrImpulses.bAtTargetPos

//NOT sv_MoldHeightEndpoints.bPositionForStepReached
;#END_EDIT_BLOCK
END_TRANSITION

GO_ON_TRANSITION Trans75 FROM Step50 TO S_Stop :=  #BEGIN_EDIT_BLOCK
TRUE
;#END_EDIT_BLOCK
END_TRANSITION

TRANSITION Trans60 FROM S_TryAgain TO S_MoldClose :=  #BEGIN_EDIT_BLOCK
TRUE
;#END_EDIT_BLOCK
END_TRANSITION

TRANSITION Trans57 FROM S_TryAgain TO S_Done :=  #BEGIN_EDIT_BLOCK
FALSE
;#END_EDIT_BLOCK
END_TRANSITION

GO_ON_TRANSITION Trans73 FROM S_Done TO S_Restart :=  #BEGIN_EDIT_BLOCK
TRUE
;#END_EDIT_BLOCK
END_TRANSITION

TRANSITION Trans71 FROM S_TryAgain TO S_Stop :=  #BEGIN_EDIT_BLOCK
FALSE
;#END_EDIT_BLOCK
END_TRANSITION

GO_ON_TRANSITION Trans72 FROM S_Stop TO S_Restart :=  #BEGIN_EDIT_BLOCK
TRUE
;#END_EDIT_BLOCK
END_TRANSITION

TRANSITION Trans74 FROM S_Restart TO START :=  #BEGIN_EDIT_BLOCK
TRUE
;#END_EDIT_BLOCK
END_TRANSITION

(* end IecGraph-Code *)
(* sfc-code *)

(* stand alone actions *)
ACTION aPreparAdjustment: #BEGIN_EDIT_BLOCK
bReady := FALSE;
bSuccess := FALSE;

IF sv_TraceLevel.bApplication THEN
    fbDebugTrace(sText := 'StretchToggleLever: start');
END_IF;

;#END_EDIT_BLOCK END_ACTION (*aPreparAdjustment*)
ACTION aCloseMold: #BEGIN_EDIT_BLOCK
// Start the mold close movement

IF sv_TraceLevel.bApplication THEN
    fbDebugTrace(sText := 'StretchToggleLever: closing Mold');
END_IF;

evStartRequestData.DeviceId := DeviceIdMold;
evStartRequestData.MoveDir := cMoveFwd;
evStartRequestData.MoveId := cMoveFwdForMHAdjustSetup;
SET_EVENT(evStartRequest, evStartRequestData);

;#END_EDIT_BLOCK END_ACTION (*aCloseMold*)
ACTION aCheckMoldClosed: #BEGIN_EDIT_BLOCK
//Check the status of mold close movement
// - Finished
// - PositionReached
fbCheckReady(DeviceId := DeviceIdMold,
             bReady => bMoldCloseReady);
fbCheckPosReached(DeviceId := DeviceIdMold,
                  MoveDir := cMoveFwd,
                  MoveId := cMoveFwdForMHAdjustSetup,
                  bPosReached => bMoldClosed);

;#END_EDIT_BLOCK END_ACTION (*aCheckMoldClosed*)
ACTION aOpenMold: #BEGIN_EDIT_BLOCK
// Start the mold open movement until protect step
IF sv_TraceLevel.bApplication THEN
    fbDebugTrace(sText := 'StretchToggleLever: opening Mold');
END_IF;

sv_bOpenMHUntilProtectStep := TRUE;

evStartRequestData.DeviceId := DeviceIdMold;
evStartRequestData.MoveDir := cMoveBwd;
evStartRequestData.MoveId := cMoveBwdForMHAdjustSetup;
SET_EVENT(evStartRequest, evStartRequestData);

;#END_EDIT_BLOCK END_ACTION (*aOpenMold*)
ACTION aCheckMoldOpen: #BEGIN_EDIT_BLOCK
// MoldHeightAdjustN.ABAdjustForceOpenLoop.paRun.aCheckMoldOpen.Check the status of mold open movement
// - Finished
// - PositionReached

fbCheckReady(DeviceId := DeviceIdMold,
             bReady => bMoldOpenReady);
fbCheckPosReached(DeviceId := DeviceIdMold,
                  MoveDir := cMoveBwd,
                  MoveId := cMoveBwdForMHAdjustSetup,
                  bPosReached => bMoldOpen);

;#END_EDIT_BLOCK END_ACTION (*aCheckMoldOpen*)
(* end sfc-code *)

END_ALGORITHM

END_ALGORITHM_BLOCK

#END_OF_IEC_PART

@Puma @IecEditor 6 30 @Pou 25
@@@BEG_Comment@@@
@h    ! WARNING !
@h    The Kemro K2 system (including software) only meets category B according to EN 954-1,
@h    thus it is not intended for usage in safety-relevant control applications in the field
@h    of personal safety (e.g. emergency stop).
@h    To implement potentially necessary safety-relevant control tasks, always use additional
@h    external safety devices that are intended for the particular purpose, and meet the necessary
@h    functional safety.
@h    For further information see EN 954-1 (EN ISO 13849-1) and/or the K2-x00 user manual, chapter
@h    "CE conformity, directives and standards".

Helper for mold height adjustment
try to stretch the toggle lever
if not possible move backward a defined pos
@@@END_Comment@@@

@BEG_Contents

@BEG_Func
@RT(17)FuncTreeContainer
2
@Var @RT(9)SET_ALARM @RT(0) @T @F @DT @RT(0) @RT(0) @T @T @UNKNOWN 0 @F
@F @F
@T
@BEG_Attrib
0 @RT(0) @RT(0)
@END_Attrib
1 1 @F @F @F @F

@Var @RT(24)REAL_TO_FORMATTED_STRING @RT(0) @T @F @DT @RT(0) @RT(0) @T @T @UNKNOWN 0 @F
@F @F
@T
@BEG_Attrib
0 @RT(0) @RT(0)
@END_Attrib
1 1 @F @F @F @F

@END_Func

@BEG_Const
@RT(18)ConstTreeContainer
0
@END_Const

@BEG_Export

@BEG_Kind
@ALGORITHM_BLOCK @RT(26)ABAdjustStretchToggleLever @STRUCTURED_TEXT
@RT(0) @RT(0) @RT(0)
@END_Kind

@BEG_Dcl
@RT(16)DclTreeContainer
5
@Var @RT(14)evStartRequest @RT(0) @T @T @DERIVED 0 @T @T @DT @RT(15)tevStartRequest @RT(0) @T @T @UNKNOWN 0 @F
@F @F
@T
@BEG_Attrib
3 @RT(0) @RT(0) @RT(0)
@END_Attrib
1 7 @F @F @F @F

@Var @RT(13)sv_TraceLevel @RT(0) @T @T @RENAMED 0 @T @T @DT @RT(12)tsTraceLevel @RT(0) @T @T @UNKNOWN 0 @F
@F @F
@T
@BEG_Attrib
3 @RT(0) @RT(0) @RT(0)
@END_Attrib
1 8 @F @F @F @F

@Var @RT(12)fbDebugTrace @RT(0) @T @T @DERIVED 0 @T @T @DT @RT(12)FBDebugTrace @RT(0) @T @T @UNKNOWN 0 @F
@F @F
@T
@BEG_Attrib
3 @RT(0) @RT(0) @RT(0)
@END_Attrib
1 0 @F @F @F @F

@Var @RT(25)erMoldHeightAdjustAborted @RT(0) @T @T @RENAMED 0 @T @T @DT @RT(5)ALARM @RT(0) @T @T @BASIC 0 @F
@F @F
@T
@BEG_Attrib
3 @RT(0) @RT(0) @RT(0)
@END_Attrib
1 7 @F @F @F @F

@Var @RT(26)sv_bOpenMHUntilProtectStep @RT(0) @T @T @RENAMED 0 @T @T @DT @RT(4)BOOL @RT(0) @T @T @BASIC 0 @F
@F @F
@T
@BEG_Attrib
3 @RT(0) @RT(0) @RT(0)
@END_Attrib
1 8 @F @F @F @F

@END_Dcl

@END_Export

@BEG_Body

1

@BEG_Export

@BEG_Algo
@ALGORITHM @RT(4)aRun @SEQUENTIAL_FLOW_CHART
@RT(0) @RT(0) @RT(0) @F @F
@END_Algo

@BEG_Dcl
@RT(16)DclTreeContainer
18
@Var @RT(5)bStop @RT(0) @T @F @DT @RT(4)BOOL @RT(0) @T @T @BASIC 0 @F
@F @F
@T
@BEG_Attrib
3 @RT(0) @RT(0) @RT(0)
@END_Attrib
1 1 @F @F @F @F

@Var @RT(12)DeviceIdMold @RT(0) @T @T @DERIVED 0 @T @T @DT @RT(10)tsDeviceId @RT(0) @T @T @UNKNOWN 0 @F
@F @F
@T
@BEG_Attrib
3 @RT(0) @RT(0) @RT(0)
@END_Attrib
1 1 @F @F @F @F

@Var @RT(18)DeviceIdMoldHeight @RT(0) @T @T @DERIVED 0 @T @T @DT @RT(10)tsDeviceId @RT(0) @T @T @UNKNOWN 0 @F
@F @F
@T
@BEG_Attrib
3 @RT(0) @RT(0) @RT(0)
@END_Attrib
1 1 @F @F @F @F

@Var @RT(12)bUseImpulses @RT(0) @T @F @DT @RT(4)BOOL @RT(0) @T @T @BASIC 0 @F
@F @F
@T
@BEG_Attrib
3 @RT(0) @RT(62)TRUE: count impulses in bwd movement FALSE: timed bwd movement @RT(0)
@END_Attrib
1 1 @F @F @F @F

@Var @RT(9)iImpulses @RT(0) @T @F @DT @RT(5)UDINT @RT(0) @T @T @BASIC 0 @F
@F @F
@T
@BEG_Attrib
3 @RT(0) @RT(47)impulses to move backward if mold can not close @RT(0)
@END_Attrib
1 1 @F @F @F @F

@Var @RT(5)dTime @RT(0) @T @F @DT @RT(4)TIME @RT(0) @T @T @BASIC 0 @F
@F @F
@T
@BEG_Attrib
3 @RT(0) @RT(43)time to move backward if mold can not close @RT(0)
@END_Attrib
1 1 @F @F @F @F

@Var @RT(6)bReady @RT(0) @T @F @DT @RT(4)BOOL @RT(0) @T @T @BASIC 0 @F
@F @F
@T
@BEG_Attrib
3 @RT(0) @RT(38)movement stopped with error or success @RT(0)
@END_Attrib
1 3 @F @F @F @F

@Var @RT(8)bSuccess @RT(0) @T @F @DT @RT(4)BOOL @RT(0) @T @T @BASIC 0 @F
@F @F
@T
@BEG_Attrib
3 @RT(0) @RT(38)if the toggle lever could be stretched @RT(0)
@END_Attrib
1 3 @F @F @F @F

@Var @RT(9)bMoldOpen @RT(0) @T @F @DT @RT(4)BOOL @RT(0) @T @T @BASIC 0 @F
@F @F
@T
@BEG_Attrib
3 @RT(0) @RT(0) @RT(0)
@END_Attrib
1 0 @F @F @F @F

@Var @RT(12)fbCheckReady @RT(0) @T @T @DERIVED 0 @T @T @DT @RT(12)FBCheckReady @RT(0) @T @T @UNKNOWN 0 @F
@F @F
@T
@BEG_Attrib
3 @RT(0) @RT(0) @RT(0)
@END_Attrib
1 0 @F @F @F @F

@Var @RT(17)fbCheckPosReached @RT(0) @T @T @DERIVED 0 @T @T @DT @RT(17)FBCheckPosReached @RT(0) @T @T @UNKNOWN 0 @F
@F @F
@T
@BEG_Attrib
3 @RT(0) @RT(0) @RT(0)
@END_Attrib
1 0 @F @F @F @F

@Var @RT(18)evStartRequestData @RT(0) @T @T @DERIVED 0 @T @T @DT @RT(19)tevStartRequestData @RT(0) @T @T @UNKNOWN 0 @F
@F @F
@T
@BEG_Attrib
3 @RT(0) @RT(0) @RT(0)
@END_Attrib
1 0 @F @F @F @F

@Var @RT(11)bMoldClosed @RT(0) @T @F @DT @RT(4)BOOL @RT(0) @T @T @BASIC 0 @F
@F @F
@T
@BEG_Attrib
3 @RT(0) @RT(0) @RT(0)
@END_Attrib
1 0 @F @F @F @F

@Var @RT(15)bMoldCloseReady @RT(0) @T @F @DT @RT(4)BOOL @RT(0) @T @T @BASIC 0 @F
@F @F
@T
@BEG_Attrib
3 @RT(0) @RT(0) @RT(0)
@END_Attrib
1 0 @F @F @F @F

@Var @RT(14)bMoldOpenReady @RT(0) @T @F @DT @RT(4)BOOL @RT(0) @T @T @BASIC 0 @F
@F @F
@T
@BEG_Attrib
3 @RT(0) @RT(0) @RT(0)
@END_Attrib
1 0 @F @F @F @F

@Var @RT(6)fbStop @RT(0) @T @T @DERIVED 0 @T @T @DT @RT(6)FBStop @RT(0) @T @T @UNKNOWN 0 @F
@F @F
@T
@BEG_Attrib
3 @RT(0) @RT(0) @RT(0)
@END_Attrib
1 0 @F @F @F @F

@Var @RT(20)dWaitAfterCloseDelay @RT(0) @T @F @DT @RT(4)TIME @RT(0) @T @T @BASIC 0 @F
@F @F
@T
@BEG_Attrib
3 @RT(7)t#100ms @RT(0) @RT(0)
@END_Attrib
1 0 @F @F @F @F

@Var @RT(20)fbMoveTimeOrImpulses @RT(0) @T @T @DERIVED 0 @T @T @DT @RT(22)FBMoveMHTimeOrImpulses @RT(0) @T @T @UNKNOWN 0 @F
@F @F
@T
@BEG_Attrib
3 @RT(0) @RT(0) @RT(0)
@END_Attrib
1 0 @F @F @F @F

@END_Dcl

@END_Export

@BEG_SfcBody
68 51 77

@BEG_SfcData 2
@StepSeq @RT(4)sseq @F 1
@Loop @RT(4)loop @F 2
@StepSeq @RT(3)seq @F 5
@Step @RT(5)START @F @T @F @F @RT(0) @F
@AcbCont @RT(7)unnamed @F 1
@Acb @RT(17)aPreparAdjustment @F @F @RT(1)P @RT(0) @F @F @T @F

@Trans @RT(6)TStart @F @T @F @F @T @T @TL(2)
TRUE

@RT(6)Trans1 @F
@Loop @RT(4)loop @F 2
@StepSeq @RT(3)seq @F 9
@Step @RT(11)S_MoldClose @F @F @F @F @RT(0) @F
@AcbCont @RT(7)unnamed @F 2
@Acb @RT(10)aCloseMold @F @F @RT(1)P @RT(0) @F @F @T @F
@Acb @RT(16)aCheckMoldClosed @F @F @RT(1)N @RT(0) @F @F @T @F

@AltBranch @RT(3)alt @F 2
@TransSeq @RT(4)tseq @F 3
@Trans @RT(15)TMoldCloseReady @F @T @F @F @T @T @TL(2)
S_MoldClose.T >= dWaitAfterCloseDelay AND bMoldCloseReady

@RT(7)Trans35 @F
@Step @RT(6)Step35 @F @F @F @F @RT(0) @F
@AcbCont @RT(7)unnamed @F 0

@AltBranch @RT(3)alt @F 2
@TransSeq @RT(4)tseq @F 1
@Trans @RT(7)Trans54 @F @T @F @F @T @F @TL(2)
NOT bMoldClosed

@RT(7)Trans54 @F

@TransSeq @RT(4)tseq @F 2
@Trans @RT(11)TMoldClosed @F @T @F @F @T @F @TL(4)
bMoldClosed
// mold could be closed,
// our part is done

@RT(7)Trans55 @F
@Goto @RT(6)S_Done @F @F

@TransSeq @RT(4)tseq @F 2
@Trans @RT(14)TStopMoldClose @F @T @F @F @T @T @TL(2)
S_MoldClose.T >= dWaitAfterCloseDelay AND bStop

@RT(7)Trans36 @F
@Goto @RT(6)S_Stop @F @F

@Step @RT(10)S_OpenMold @F @F @F @F @RT(0) @F
@AcbCont @RT(7)unnamed @F 2
@Acb @RT(9)aOpenMold @F @F @RT(1)P @RT(0) @F @F @T @F
@Acb @RT(14)aCheckMoldOpen @F @F @RT(1)N @RT(0) @F @F @T @F

@AltBranch @RT(3)alt @F 2
@TransSeq @RT(4)tseq @F 1
@Trans @RT(11)TMoldIsOpen @F @T @F @F @T @T @TL(2)
bMoldOpenReady

@RT(7)Trans20 @F

@TransSeq @RT(4)tseq @F 2
@Trans @RT(7)Trans76 @F @T @F @F @T @T @TL(2)
bStop

@RT(7)Trans76 @F
@Goto @RT(6)S_Stop @F @F

@Step @RT(7)S_MHBwd @F @F @F @F @RT(0) @F
@AcbCont @RT(7)unnamed @F 1
@Acb @RT(8)Action66 @F @T @RT(1)N @RT(0) @F @F @T @TL(3)
fbMoveTimeOrImpulses(bUseImpulses := bUseImpulses, dTime := dTime, iImpulses := iImpulses,
                    DeviceId := DeviceIdMoldHeight, MoveDir := cMoveBwd, MoveId := cMoveBwd);

@F

@AltBranch @RT(3)alt @F 2
@TransSeq @RT(4)tseq @F 1
@Trans @RT(15)TAdjustBwdReady @F @T @F @F @T @T @TL(6)
fbMoveTimeOrImpulses.bDone

//AND
//fbMoveTimeOrImpulses.
//bAdjustBwdReady

@RT(7)Trans38 @F

@TransSeq @RT(4)tseq @F 2
@Trans @RT(11)TStopAdjBwd @F @T @F @F @T @T @TL(5)
bStop

//OR
//(fbMoveTimeOrImpulses.bDone AND NOT fbMoveTimeOrImpulses.bAtTargetPos)

@RT(7)Trans39 @F
@Goto @RT(6)S_Stop @F @F

@Step @RT(6)Step26 @F @F @F @F @RT(0) @F
@AcbCont @RT(7)unnamed @F 0

@AltBranch @RT(3)alt @F 2
@TransSeq @RT(4)tseq @F 1
@Trans @RT(16)AdjBwdPosReached @F @T @F @F @T @F @TL(4)
fbMoveTimeOrImpulses.bAtTargetPos

//sv_MoldHeightEndpoints.bPositionForStepReached

@RT(6)Trans9 @F

@TransSeq @RT(4)tseq @F 4
@Trans @RT(19)AdjBwdPosNotReached @F @T @F @F @T @F @TL(4)
NOT fbMoveTimeOrImpulses.bAtTargetPos

//NOT sv_MoldHeightEndpoints.bPositionForStepReached

@RT(7)Trans40 @F
@Step @RT(6)Step50 @F @F @F @F @RT(0) @F
@AcbCont @RT(7)unnamed @F 1
@Acb @RT(8)Action67 @F @T @RT(1)N @RT(0) @F @F @T @TL(3)
SET_ALARM(erMoldHeightAdjustAborted);
//FIXME: maybe use different alarm

@F

@Trans @RT(7)Trans75 @F @T @F @F @T @F @TL(2)
TRUE

@RT(7)Trans75 @F
@Goto @RT(6)S_Stop @F @F

@Step @RT(10)S_TryAgain @F @F @F @F @RT(0) @F
@AcbCont @RT(7)unnamed @F 0

@Trans @RT(7)Trans60 @F @T @T @T @T @T @TL(2)
TRUE

@RT(7)Trans60 @F

@AltBranch @RT(3)alt @F 2
@TransSeq @RT(4)tseq @F 3
@Trans @RT(7)Trans57 @F @T @F @F @T @T @TL(2)
FALSE

@RT(7)Trans57 @F
@Step @RT(6)S_Done @F @F @T @F @RT(0) @F
@AcbCont @RT(7)unnamed @F 1
@Acb @RT(5)aDone @F @T @RT(1)P @RT(0) @F @F @T @TL(3)
//toggle lever is stretched
bSuccess := TRUE;

@F

@Trans @RT(7)Trans73 @F @T @F @F @T @F @TL(2)
TRUE

@RT(7)Trans73 @F

@TransSeq @RT(4)tseq @F 3
@Trans @RT(7)Trans71 @F @T @F @F @T @T @TL(2)
FALSE

@RT(7)Trans71 @F
@Step @RT(6)S_Stop @F @F @T @F @RT(0) @F
@AcbCont @RT(7)unnamed @F 1
@Acb @RT(7)aFailed @F @T @RT(1)N @RT(0) @F @F @T @TL(2)
bSuccess := FALSE;

@F

@Trans @RT(7)Trans72 @F @T @F @F @T @F @TL(2)
TRUE

@RT(7)Trans72 @F

@Step @RT(9)S_Restart @F @F @F @F @RT(0) @F
@AcbCont @RT(7)unnamed @F 1
@Acb @RT(5)AStop @F @T @RT(1)P @RT(0) @F @F @T @TL(10)
//stop active movement
IF bStop THEN
    fbStop(DeviceId := DeviceIdMold);
    fbStop(DeviceId := DeviceIdMoldHeight);
END_IF;

sv_bOpenMHUntilProtectStep :=FALSE;

bReady := TRUE;

@F

@Trans @RT(7)Trans74 @F @T @T @T @T @T @TL(2)
TRUE

@RT(7)Trans74 @F

@END_SfcData
@SaActions 5
@SaText @RT(17)aPreparAdjustment 1 @TL(8)
bReady := FALSE;
bSuccess := FALSE;

IF sv_TraceLevel.bApplication THEN
    fbDebugTrace(sText := 'StretchToggleLever: start');
END_IF;

@SaText @RT(10)aCloseMold 1 @TL(13)
// Start the mold close movement

IF sv_TraceLevel.bApplication THEN
    fbDebugTrace(sText := 'StretchToggleLever: closing Mold');
END_IF;

evStartRequestData.DeviceId := DeviceIdMold;
evStartRequestData.MoveDir := cMoveFwd;
evStartRequestData.MoveId := cMoveFwdForMHAdjustSetup;
SET_EVENT(evStartRequest, evStartRequestData);

@SaText @RT(16)aCheckMoldClosed 1 @TL(10)
//Check the status of mold close movement
// - Finished
// - PositionReached
fbCheckReady(DeviceId := DeviceIdMold,
             bReady => bMoldCloseReady);
fbCheckPosReached(DeviceId := DeviceIdMold,
                  MoveDir := cMoveFwd,
                  MoveId := cMoveFwdForMHAdjustSetup,
                  bPosReached => bMoldClosed);

@SaText @RT(9)aOpenMold 1 @TL(12)
// Start the mold open movement until protect step
IF sv_TraceLevel.bApplication THEN
    fbDebugTrace(sText := 'StretchToggleLever: opening Mold');
END_IF;

sv_bOpenMHUntilProtectStep := TRUE;

evStartRequestData.DeviceId := DeviceIdMold;
evStartRequestData.MoveDir := cMoveBwd;
evStartRequestData.MoveId := cMoveBwdForMHAdjustSetup;
SET_EVENT(evStartRequest, evStartRequestData);

@SaText @RT(14)aCheckMoldOpen 1 @TL(11)
// MoldHeightAdjustN.ABAdjustForceOpenLoop.paRun.aCheckMoldOpen.Check the status of mold open movement
// - Finished
// - PositionReached

fbCheckReady(DeviceId := DeviceIdMold,
             bReady => bMoldOpenReady);
fbCheckPosReached(DeviceId := DeviceIdMold,
                  MoveDir := cMoveBwd,
                  MoveId := cMoveBwdForMHAdjustSetup,
                  bPosReached => bMoldOpen);

@SaTrans 0
@SaExits 0
@END_SfcBody

@@@BEG_Comment@@@
@TL(9)
Stretch the toggle lever:

try to close mold
if not possible (standstill before pos 0)
  open mold again
  move mold height backward
  try again

mold close possible -> done
@@@END_Comment@@@
@END_Body

@END_Contents
